KUKA KRL program: EPS_2_25856_SANMH_A_20250918023512.src

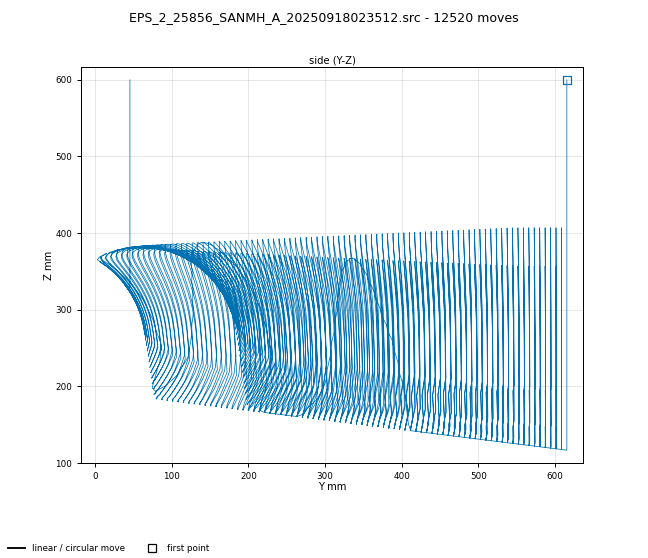
[picture p0: tool path of EPS_2_25856_SANMH_A_20250918023512.src, 12520 of 12522 moves have a stored position in this frame; points joined in program order, loops and branches not executed]
&ACCESS RVP
&REL 4
&COMMENT QRS 19112012
&PARAM EDITMASK = *
DEF PART()
EXT BAS (BAS_COMMAND :IN,REAL :IN )
INT I
BAS (#INITMOV,0 )

;KUKA QRS Post kuka4.cps  Date:22-06-2017 !

File_ID=2850

QRS_PRE_INIT()

;Init var - Until changes are made in qrs_pre_init
Outlet_Square_prg=0
Inlet_1_Square_prg=0
Inlet_2_Square_prg=0
Inlet_3_Square_prg=0
Inlet_4_Square_prg=0
Inlet_5_Square_prg=0

Outlet_1={X 0.000, Y 546.330, Z 306.500, B 0.000, E1 0.000 }
Inlet_1={X 0.000, Y 549.890, Z 256.500, B 0.000, E1 218.000 }
Outlet_1_type=201
Inlet_1_type=201
;QRS#1=Sidecore dimensions
;QRS#2=200-8" PVC SDR 35
;QRS#3=200-8" PVC SDR 35
;QRS#4=
;QRS#5=
;QRS#6=
;QRS#7=
;QRS#8=
;QRS#9=12-08 PSX
;QRS#10=12-08 PSX
;QRS#11=
;QRS#12=
;QRS#13=
;QRS#14=
;QRS#15=
;QRS#16=1220x127x686 2,25'
;QRS#17=EPS Height
;QRS#18=407
;QRS#19=*
;QRS#20= UPDATED VERSION 22-06-2017
;QRS#21=*
Outlet_Square=0100
Inlet_1_Square=0100
Inlet_2_Square=0
Inlet_3_Square=0
Inlet_4_Square=0
Inlet_5_Square=0
Mill_Square=1
Outlet_Square_Prg=204
Inlet_1_Square_prg=204

QRS_INIT()

$ADVANCE=5

; T1
PTP {E1 173.606,E2 173.606}
PTP {X 0,Y 615.506,A -85,B 0,C 180,E1 173.606,E2 173.606,E3 0,E4 0,E5 0,E6 0}
QRS_SPEED_INIT()
LIN {X 0,Y 615.506,Z 600,A -85,B 0,C 180,E1 173.606,E2 173.606,E3 0,E4 0,E5 0,E6 0} C_VEL
LIN {X 0,Y 615.506,Z 126.869,A -85,B 0,C 180,E1 173.606,E2 173.606} C_VEL
LIN {X 0,Y 615.506,Z 118.698,A -85,B 0,C 180,E1 173.606,E2 173.606} C_VEL
LIN {X 0,Y 615.487,Z 116.698,A -85,B 0,C 180,E1 173.42,E2 173.42} C_VEL
LIN {X 0,Y 615.471,Z 116.691,A -85,B 0,C 180,E1 170.801,E2 170.801} C_VEL
LIN {X 0,Y 615.488,Z 116.684,A -85,B 0,C 180,E1 168.14,E2 168.14} C_VEL
LIN {X 0,Y 615.489,Z 116.702,A -85,B 0,C 180,E1 165.451,E2 165.451} C_VEL
LIN {X 0,Y 615.476,Z 116.686,A -85,B 0,C 180,E1 162.73,E2 162.73} C_VEL
LIN {X 0,Y 615.48,Z 116.692,A -85,B 0,C 180,E1 159.967,E2 159.967} C_VEL
LIN {X 0,Y 615.492,Z 116.701,A -85,B 0,C 180,E1 157.652,E2 157.652} C_VEL
LIN {X 0,Y 615.473,Z 116.688,A -85,B 0,C 180,E1 155.008,E2 155.008} C_VEL
LIN {X 0,Y 615.481,Z 116.684,A -85,B 0,C 180,E1 152.823,E2 152.823} C_VEL
LIN {X 0,Y 615.482,Z 116.69,A -85,B 0,C 180,E1 150.206,E2 150.206} C_VEL
LIN {X 0,Y 615.48,Z 116.695,A -85,B 0,C 180,E1 147.543,E2 147.543} C_VEL
LIN {X 0,Y 615.475,Z 116.687,A -85,B 0,C 180,E1 145.185,E2 145.185} C_VEL
LIN {X 0,Y 615.493,Z 116.682,A -85,B 0,C 180,E1 142.759,E2 142.759} C_VEL
LIN {X 0,Y 615.494,Z 116.699,A -85,B 0,C 180,E1 139.91,E2 139.91} C_VEL
LIN {X 0,Y 615.488,Z 116.683,A -85,B 0,C 180,E1 136.952,E2 136.952} C_VEL
LIN {X 0,Y 615.49,Z 116.699,A -85,B 0,C 180,E1 133.998,E2 133.998} C_VEL
LIN {X 0,Y 615.487,Z 116.683,A -85,B 0,C 180,E1 131.095,E2 131.095} C_VEL
LIN {X 0,Y 615.487,Z 116.697,A -85,B 0,C 180,E1 128.068,E2 128.068} C_VEL
LIN {X 0,Y 615.473,Z 116.688,A -85,B 0,C 180,E1 125.616,E2 125.616} C_VEL
LIN {X 0,Y 615.487,Z 116.683,A -85,B 0,C 180,E1 123.236,E2 123.236} C_VEL
LIN {X 0,Y 615.481,Z 116.688,A -85,B 0,C 180,E1 120.92,E2 120.92} C_VEL
LIN {X 0,Y 615.497,Z 116.699,A -85,B 0,C 180,E1 118.453,E2 118.453} C_VEL
LIN {X 0,Y 615.485,Z 116.683,A -85,B 0,C 180,E1 115.569,E2 115.569} C_VEL
LIN {X 0,Y 615.482,Z 116.694,A -85,B 0,C 180,E1 112.844,E2 112.844} C_VEL
LIN {X 0,Y 615.488,Z 116.702,A -85,B 0,C 180,E1 110.558,E2 110.558} C_VEL
LIN {X 0,Y 615.478,Z 116.687,A -85,B 0,C 180,E1 107.957,E2 107.957} C_VEL
LIN {X 0,Y 615.479,Z 116.689,A -85,B 0,C 180,E1 105.226,E2 105.226} C_VEL
LIN {X 0,Y 615.485,Z 116.696,A -85,B 0,C 180,E1 102.53,E2 102.53} C_VEL
LIN {X 0,Y 615.493,Z 116.681,A -85,B 0,C 180,E1 99.862,E2 99.862} C_VEL
LIN {X 0,Y 615.48,Z 116.693,A -85,B 0,C 180,E1 97.215,E2 97.215} C_VEL
LIN {X 0,Y 615.48,Z 116.694,A -85,B 0,C 180,E1 94.584,E2 94.584} C_VEL
LIN {X 0,Y 615.5,Z 116.68,A -85,B 0,C 180,E1 91.963,E2 91.963} C_VEL
LIN {X 0,Y 615.48,Z 116.693,A -85,B 0,C 180,E1 89.345,E2 89.345} C_VEL
LIN {X 0,Y 615.48,Z 116.693,A -85,B 0,C 180,E1 86.727,E2 86.727} C_VEL
LIN {X 0,Y 615.498,Z 116.68,A -85,B 0,C 180,E1 84.101,E2 84.101} C_VEL
LIN {X 0,Y 615.481,Z 116.694,A -85,B 0,C 180,E1 81.463,E2 81.463} C_VEL
LIN {X 0,Y 615.477,Z 116.692,A -85,B 0,C 180,E1 78.806,E2 78.806} C_VEL
LIN {X 0,Y 615.483,Z 116.685,A -85,B 0,C 180,E1 76.067,E2 76.067} C_VEL
LIN {X 0,Y 615.494,Z 116.699,A -85,B 0,C 180,E1 73.413,E2 73.413} C_VEL
LIN {X 0,Y 615.485,Z 116.685,A -85,B 0,C 180,E1 70.662,E2 70.662} C_VEL
LIN {X 0,Y 615.476,Z 116.819,A -85,B 0,C 180,E1 69.966,E2 69.966} C_VEL
LIN {X 0,Y 615.473,Z 131.445,A -85,B 0,C 180,E1 67.404,E2 67.404} C_VEL
LIN {X 0,Y 615.472,Z 146.428,A -85,B 0,C 180,E1 64.808,E2 64.808} C_VEL
LIN {X 0,Y 615.434,Z 253.444,A -85,B 0,C 180,E1 63.534,E2 63.534} C_VEL
LIN {X 0,Y 615.441,Z 266.025,A -85,B 0,C 180,E1 63.256,E2 63.256} C_VEL
LIN {X 0,Y 615.475,Z 279.168,A -85,B 0,C 180,E1 62.822,E2 62.822} C_VEL
LIN {X 0,Y 615.472,Z 291.37,A -85,B 0,C 180,E1 62.269,E2 62.269} C_VEL
LIN {X 0,Y 615.477,Z 302.53,A -85,B 0,C 180,E1 61.617,E2 61.617} C_VEL
LIN {X 0,Y 615.5,Z 312.724,A -85,B 0,C 180,E1 60.875,E2 60.875} C_VEL
LIN {X 0,Y 615.498,Z 322.222,A -85,B 0,C 180,E1 60.021,E2 60.021} C_VEL
LIN {X 0,Y 615.497,Z 330.704,A -85,B 0,C 180,E1 59.08,E2 59.08} C_VEL
LIN {X 0,Y 615.498,Z 337.512,A -85,B 0,C 180,E1 58.153,E2 58.153} C_VEL
LIN {X 0,Y 615.495,Z 343.437,A -85,B 0,C 180,E1 57.154,E2 57.154} C_VEL
LIN {X 0,Y 615.495,Z 348.788,A -85,B 0,C 180,E1 55.978,E2 55.978} C_VEL
LIN {X 0,Y 615.497,Z 352.664,A -85,B 0,C 180,E1 54.786,E2 54.786} C_VEL
LIN {X 0,Y 615.494,Z 355.18,A -85,B 0,C 180,E1 53.575,E2 53.575} C_VEL
LIN {X 0,Y 615.496,Z 356.068,A -85,B 0,C 180,E1 52.758,E2 52.758} C_VEL
LIN {X 0,Y 615.494,Z 356.387,A -85,B 0,C 180,E1 51.931,E2 51.931} C_VEL
LIN {X 0,Y 615.495,Z 355.914,A -85,B 0,C 180,E1 50.936,E2 50.936} C_VEL
LIN {X 0,Y 615.496,Z 354.47,A -85,B 0,C 180,E1 49.909,E2 49.909} C_VEL
LIN {X 0,Y 615.494,Z 352.075,A -85,B 0,C 180,E1 48.904,E2 48.904} C_VEL
LIN {X 0,Y 615.497,Z 348.737,A -85,B 0,C 180,E1 47.918,E2 47.918} C_VEL
LIN {X 0,Y 615.498,Z 343.434,A -85,B 0,C 180,E1 46.756,E2 46.756} C_VEL
LIN {X 0,Y 615.494,Z 336.828,A -85,B 0,C 180,E1 45.655,E2 45.655} C_VEL
LIN {X 0,Y 615.495,Z 329.928,A -85,B 0,C 180,E1 44.735,E2 44.735} C_VEL
LIN {X 0,Y 615.498,Z 321.427,A -85,B 0,C 180,E1 43.808,E2 43.808} C_VEL
LIN {X 0,Y 615.499,Z 311.77,A -85,B 0,C 180,E1 42.96,E2 42.96} C_VEL
LIN {X 0,Y 615.47,Z 301.331,A -85,B 0,C 180,E1 42.215,E2 42.215} C_VEL
LIN {X 0,Y 615.466,Z 291.064,A -85,B 0,C 180,E1 41.625,E2 41.625} C_VEL
LIN {X 0,Y 615.486,Z 279.307,A -85,B 0,C 180,E1 41.094,E2 41.094} C_VEL
LIN {X 0,Y 615.456,Z 266.543,A -85,B 0,C 180,E1 40.669,E2 40.669} C_VEL
LIN {X 0,Y 615.445,Z 253.621,A -85,B 0,C 180,E1 40.379,E2 40.379} C_VEL
LIN {X 0,Y 615.497,Z 146.435,A -85,B 0,C 180,E1 39.104,E2 39.104} C_VEL
LIN {X 0,Y 615.48,Z 130.975,A -85,B 0,C 180,E1 36.425,E2 36.425} C_VEL
LIN {X 0,Y 615.465,Z 116.691,A -85,B 0,C 180,E1 33.9,E2 33.9} C_VEL
LIN {X 0,Y 615.491,Z 116.688,A -85,B 0,C 180,E1 31.086,E2 31.086} C_VEL
LIN {X 0,Y 615.475,Z 116.697,A -85,B 0,C 180,E1 28.447,E2 28.447} C_VEL
LIN {X 0,Y 615.472,Z 116.687,A -85,B 0,C 180,E1 25.716,E2 25.716} C_VEL
LIN {X 0,Y 615.483,Z 116.701,A -85,B 0,C 180,E1 22.844,E2 22.844} C_VEL
LIN {X 0,Y 615.46,Z 116.695,A -85,B 0,C 180,E1 20.549,E2 20.549} C_VEL
LIN {X 0,Y 615.464,Z 116.689,A -85,B 0,C 180,E1 17.957,E2 17.957} C_VEL
LIN {X 0,Y 615.492,Z 116.701,A -85,B 0,C 180,E1 15.225,E2 15.225} C_VEL
LIN {X 0,Y 615.446,Z 116.694,A -85,B 0,C 180,E1 12.531,E2 12.531} C_VEL
LIN {X 0,Y 615.49,Z 116.688,A -85,B 0,C 180,E1 9.862,E2 9.862} C_VEL
LIN {X 0,Y 615.467,Z 116.698,A -85,B 0,C 180,E1 7.216,E2 7.216} C_VEL
LIN {X 0,Y 615.462,Z 116.698,A -85,B 0,C 180,E1 5.241,E2 5.241} C_VEL
LIN {X 0,Y 615.438,Z 116.694,A -85,B 0,C 180,E1 2.618,E2 2.618} C_VEL
LIN {X 0,Y 615.487,Z 116.695,A -85,B 0,C 180,E1 0,E2 0} C_VEL
LIN {X 0,Y 615.446,Z 116.698,A -85,B 0,C 180,E1 -2.618,E2 -2.618} C_VEL
LIN {X 0,Y 615.442,Z 116.699,A -85,B 0,C 180,E1 -4.585,E2 -4.585} C_VEL
LIN {X 0,Y 615.438,Z 116.699,A -85,B 0,C 180,E1 -6.558,E2 -6.558} C_VEL
LIN {X 0,Y 615.433,Z 116.699,A -85,B 0,C 180,E1 -8.538,E2 -8.538} C_VEL
LIN {X 0,Y 615.42,Z 116.698,A -85,B 0,C 180,E1 -10.853,E2 -10.853} C_VEL
LIN {X 0,Y 615.437,Z 116.699,A -85,B 0,C 180,E1 -13.203,E2 -13.203} C_VEL
LIN {X 0,Y 615.464,Z 116.7,A -85,B 0,C 180,E1 -15.906,E2 -15.906} C_VEL
LIN {X 0,Y 615.414,Z 116.7,A -85,B 0,C 180,E1 -18.649,E2 -18.649} C_VEL
LIN {X 0,Y 615.495,Z 116.7,A -85,B 0,C 180,E1 -21.432,E2 -21.432} C_VEL
LIN {X 0,Y 615.422,Z 116.698,A -85,B 0,C 180,E1 -24.275,E2 -24.275} C_VEL
LIN {X 0,Y 615.424,Z 116.698,A -85,B 0,C 180,E1 -26.447,E2 -26.447} C_VEL
LIN {X 0,Y 615.483,Z 116.696,A -85,B 0,C 180,E1 -29.407,E2 -29.407} C_VEL
LIN {X 0,Y 615.452,Z 116.694,A -85,B 0,C 180,E1 -31.688,E2 -31.688} C_VEL
LIN {X 0,Y 615.433,Z 116.696,A -85,B 0,C 180,E1 -34.026,E2 -34.026} C_VEL
LIN {X 0,Y 615.488,Z 116.701,A -85,B 0,C 180,E1 -36.936,E2 -36.936} C_VEL
LIN {X 0,Y 615.44,Z 116.694,A -85,B 0,C 180,E1 -39.754,E2 -39.754} C_VEL
LIN {X 0,Y 615.461,Z 116.698,A -85,B 0,C 180,E1 -42.356,E2 -42.356} C_VEL
LIN {X 0,Y 615.491,Z 116.688,A -85,B 0,C 180,E1 -45.069,E2 -45.069} C_VEL
LIN {X 0,Y 615.447,Z 116.693,A -85,B 0,C 180,E1 -47.643,E2 -47.643} C_VEL
LIN {X 0,Y 615.479,Z 116.699,A -85,B 0,C 180,E1 -50.249,E2 -50.249} C_VEL
LIN {X 0,Y 615.474,Z 116.688,A -85,B 0,C 180,E1 -53.066,E2 -53.066} C_VEL
LIN {X 0,Y 615.457,Z 116.69,A -85,B 0,C 180,E1 -55.304,E2 -55.304} C_VEL
LIN {X 0,Y 615.461,Z 116.695,A -85,B 0,C 180,E1 -57.674,E2 -57.674} C_VEL
LIN {X 0,Y 615.489,Z 116.687,A -85,B 0,C 180,E1 -60.593,E2 -60.593} C_VEL
LIN {X 0,Y 615.468,Z 116.688,A -85,B 0,C 180,E1 -62.959,E2 -62.959} C_VEL
LIN {X 0,Y 615.482,Z 116.7,A -85,B 0,C 180,E1 -65.727,E2 -65.727} C_VEL
LIN {X 0,Y 615.464,Z 116.819,A -85,B 0,C 180,E1 -67.065,E2 -67.065} C_VEL
LIN {X 0,Y 615.465,Z 136.769,A -85,B 0,C 180,E1 -69.706,E2 -69.706} C_VEL
LIN {X 0,Y 615.485,Z 158.666,A -85,B 0,C 180,E1 -72.558,E2 -72.558} C_VEL
LIN {X 0,Y 615.469,Z 179.888,A -85,B 0,C 180,E1 -75.281,E2 -75.281} C_VEL
LIN {X 0,Y 615.452,Z 194.297,A -85,B 0,C 180,E1 -77.112,E2 -77.112} C_VEL
LIN {X 0,Y 615.488,Z 302.807,A -85,B 0,C 180,E1 -78.41,E2 -78.41} C_VEL
LIN {X 0,Y 615.477,Z 315.331,A -85,B 0,C 180,E1 -78.681,E2 -78.681} C_VEL
LIN {X 0,Y 615.488,Z 328.619,A -85,B 0,C 180,E1 -79.113,E2 -79.113} C_VEL
LIN {X 0,Y 615.477,Z 340.471,A -85,B 0,C 180,E1 -79.639,E2 -79.639} C_VEL
LIN {X 0,Y 615.494,Z 351.988,A -85,B 0,C 180,E1 -80.303,E2 -80.303} C_VEL
LIN {X 0,Y 615.499,Z 362.336,A -85,B 0,C 180,E1 -81.049,E2 -81.049} C_VEL
LIN {X 0,Y 615.497,Z 370.807,A -85,B 0,C 180,E1 -81.794,E2 -81.794} C_VEL
LIN {X 0,Y 615.498,Z 378.603,A -85,B 0,C 180,E1 -82.619,E2 -82.619} C_VEL
LIN {X 0,Y 615.496,Z 386.2,A -85,B 0,C 180,E1 -83.608,E2 -83.608} C_VEL
LIN {X 0,Y 615.498,Z 393.202,A -85,B 0,C 180,E1 -84.759,E2 -84.759} C_VEL
LIN {X 0,Y 615.494,Z 397.85,A -85,B 0,C 180,E1 -85.743,E2 -85.743} C_VEL
LIN {X 0,Y 615.494,Z 401.397,A -85,B 0,C 180,E1 -86.727,E2 -86.727} C_VEL
LIN {X 0,Y 615.497,Z 403.232,A -85,B 0,C 180,E1 -87.382,E2 -87.382} C_VEL
LIN {X 0,Y 615.5,Z 404.607,A -85,B 0,C 180,E1 -88.037,E2 -88.037} C_VEL
LIN {X 0,Y 615.496,Z 406.173,A -85,B 0,C 180,E1 -89.345,E2 -89.345} C_VEL
LIN {X 0,Y 615.494,Z 406.389,A -85,B 0,C 180,E1 -90,E2 -90} C_VEL
LIN {X 0,Y 615.495,Z 405.58,A -85,B 0,C 180,E1 -91.308,E2 -91.308} C_VEL
LIN {X 0,Y 615.5,Z 404.608,A -85,B 0,C 180,E1 -91.963,E2 -91.963} C_VEL
LIN {X 0,Y 615.497,Z 403.234,A -85,B 0,C 180,E1 -92.617,E2 -92.617} C_VEL
LIN {X 0,Y 615.496,Z 400.351,A -85,B 0,C 180,E1 -93.6,E2 -93.6} C_VEL
LIN {X 0,Y 615.498,Z 396.443,A -85,B 0,C 180,E1 -94.584,E2 -94.584} C_VEL
LIN {X 0,Y 615.499,Z 391.407,A -85,B 0,C 180,E1 -95.569,E2 -95.569} C_VEL
LIN {X 0,Y 615.497,Z 384.87,A -85,B 0,C 180,E1 -96.583,E2 -96.583} C_VEL
LIN {X 0,Y 615.497,Z 377.136,A -85,B 0,C 180,E1 -97.545,E2 -97.545} C_VEL
LIN {X 0,Y 615.498,Z 369.049,A -85,B 0,C 180,E1 -98.371,E2 -98.371} C_VEL
LIN {X 0,Y 615.499,Z 359.172,A -85,B 0,C 180,E1 -99.198,E2 -99.198} C_VEL
LIN {X 0,Y 615.488,Z 347.988,A -85,B 0,C 180,E1 -99.945,E2 -99.945} C_VEL
LIN {X 0,Y 615.482,Z 337.031,A -85,B 0,C 180,E1 -100.527,E2 -100.527} C_VEL
LIN {X 0,Y 615.48,Z 324.496,A -85,B 0,C 180,E1 -101.04,E2 -101.04} C_VEL
LIN {X 0,Y 615.479,Z 312.083,A -85,B 0,C 180,E1 -101.401,E2 -101.401} C_VEL
LIN {X 0,Y 615.493,Z 298.491,A -85,B 0,C 180,E1 -101.651,E2 -101.651} C_VEL
LIN {X 0,Y 615.452,Z 194.304,A -85,B 0,C 180,E1 -102.887,E2 -102.887} C_VEL
LIN {X 0,Y 615.494,Z 171.936,A -85,B 0,C 180,E1 -105.735,E2 -105.735} C_VEL
LIN {X 0,Y 615.456,Z 151.013,A -85,B 0,C 180,E1 -108.435,E2 -108.435} C_VEL
LIN {X 0,Y 615.488,Z 130.785,A -85,B 0,C 180,E1 -111.08,E2 -111.08} C_VEL
LIN {X 0,Y 615.465,Z 116.689,A -85,B 0,C 180,E1 -112.978,E2 -112.978} C_VEL
LIN {X 0,Y 615.489,Z 116.689,A -85,B 0,C 180,E1 -115.715,E2 -115.715} C_VEL
LIN {X 0,Y 615.469,Z 116.696,A -85,B 0,C 180,E1 -118.447,E2 -118.447} C_VEL
LIN {X 0,Y 615.479,Z 116.684,A -85,B 0,C 180,E1 -121.084,E2 -121.084} C_VEL
LIN {X 0,Y 615.492,Z 116.701,A -85,B 0,C 180,E1 -124.021,E2 -124.021} C_VEL
LIN {X 0,Y 615.478,Z 116.685,A -85,B 0,C 180,E1 -126.935,E2 -126.935} C_VEL
LIN {X 0,Y 615.491,Z 116.698,A -85,B 0,C 180,E1 -129.749,E2 -129.749} C_VEL
LIN {X 0,Y 615.466,Z 116.692,A -85,B 0,C 180,E1 -132.354,E2 -132.354} C_VEL
LIN {X 0,Y 615.496,Z 116.683,A -85,B 0,C 180,E1 -135.067,E2 -135.067} C_VEL
LIN {X 0,Y 615.481,Z 116.697,A -85,B 0,C 180,E1 -137.92,E2 -137.92} C_VEL
LIN {X 0,Y 615.465,Z 116.691,A -85,B 0,C 180,E1 -140.248,E2 -140.248} C_VEL
LIN {X 0,Y 615.488,Z 116.687,A -85,B 0,C 180,E1 -143.063,E2 -143.063} C_VEL
LIN {X 0,Y 615.47,Z 116.693,A -85,B 0,C 180,E1 -145.977,E2 -145.977} C_VEL
LIN {X 0,Y 615.469,Z 116.688,A -85,B 0,C 180,E1 -148.313,E2 -148.313} C_VEL
LIN {X 0,Y 615.486,Z 116.683,A -85,B 0,C 180,E1 -150.593,E2 -150.593} C_VEL
LIN {X 0,Y 615.481,Z 116.698,A -85,B 0,C 180,E1 -153.555,E2 -153.555} C_VEL
LIN {X 0,Y 615.485,Z 116.684,A -85,B 0,C 180,E1 -156.443,E2 -156.443} C_VEL
LIN {X 0,Y 615.481,Z 116.698,A -85,B 0,C 180,E1 -159.444,E2 -159.444} C_VEL
LIN {X 0,Y 615.473,Z 116.686,A -85,B 0,C 180,E1 -162.042,E2 -162.042} C_VEL
LIN {X 0,Y 615.485,Z 116.691,A -85,B 0,C 180,E1 -164.774,E2 -164.774} C_VEL
LIN {X 0,Y 615.471,Z 116.695,A -85,B 0,C 180,E1 -167.469,E2 -167.469} C_VEL
LIN {X 0,Y 615.492,Z 116.682,A -85,B 0,C 180,E1 -170.138,E2 -170.138} C_VEL
LIN {X 0,Y 615.489,Z 116.695,A -85,B 0,C 180,E1 -172.784,E2 -172.784} C_VEL
LIN {X 0,Y 615.471,Z 116.692,A -85,B 0,C 180,E1 -175.415,E2 -175.415} C_VEL
LIN {X 0,Y 615.5,Z 116.68,A -85,B 0,C 180,E1 -178.037,E2 -178.037} C_VEL
LIN {X 0,Y 615.49,Z 116.696,A -85,B 0,C 180,E1 -180.654,E2 -180.654} C_VEL
LIN {X 0,Y 615.471,Z 116.692,A -85,B 0,C 180,E1 -183.273,E2 -183.273} C_VEL
LIN {X 0,Y 615.498,Z 116.681,A -85,B 0,C 180,E1 -185.898,E2 -185.898} C_VEL
LIN {X 0,Y 615.487,Z 116.698,A -85,B 0,C 180,E1 -186.58,E2 -186.58} C_VEL
LIN {X 0,Y 614.8,Z 116.838,A -85,B 0,C 180,E1 -187.126,E2 -187.126} C_VEL
LIN {X 0,Y 611.955,Z 117.252,A -85,B 0,C 180,E1 -188.012,E2 -188.012} C_VEL
LIN {X 0,Y 609.565,Z 117.562,A -85,B 0,C 180,E1 -188.725,E2 -188.725} C_VEL
LIN {X 0,Y 608.538,Z 117.679,A -85,B 0,C 180,E1 -189.274,E2 -189.274} C_VEL
LIN {X 0,Y 608.453,Z 117.688,A -85,B 0,C 180,E1 -189.461,E2 -189.461} C_VEL
LIN {X 0,Y 608.464,Z 117.688,A -85,B 0,C 180,E1 -191.999,E2 -191.999} C_VEL
LIN {X 0,Y 608.474,Z 117.692,A -85,B 0,C 180,E1 -194.72,E2 -194.72} C_VEL
LIN {X 0,Y 608.445,Z 117.688,A -85,B 0,C 180,E1 -197.476,E2 -197.476} C_VEL
LIN {X 0,Y 608.461,Z 117.694,A -85,B 0,C 180,E1 -200.274,E2 -200.274} C_VEL
LIN {X 0,Y 608.455,Z 117.696,A -85,B 0,C 180,E1 -202.476,E2 -202.476} C_VEL
LIN {X 0,Y 608.449,Z 117.694,A -85,B 0,C 180,E1 -204.571,E2 -204.571} C_VEL
LIN {X 0,Y 608.473,Z 117.685,A -85,B 0,C 180,E1 -207.207,E2 -207.207} C_VEL
LIN {X 0,Y 608.467,Z 117.692,A -85,B 0,C 180,E1 -209.972,E2 -209.972} C_VEL
LIN {X 0,Y 608.455,Z 117.692,A -85,B 0,C 180,E1 -212.522,E2 -212.522} C_VEL
LIN {X 0,Y 608.436,Z 117.69,A -85,B 0,C 180,E1 -215.278,E2 -215.278} C_VEL
LIN {X 0,Y 608.471,Z 117.69,A -85,B 0,C 180,E1 -217.746,E2 -217.746} C_VEL
LIN {X 0,Y 608.45,Z 117.693,A -85,B 0,C 180,E1 -220.329,E2 -220.329} C_VEL
LIN {X 0,Y 608.453,Z 117.687,A -85,B 0,C 180,E1 -222.959,E2 -222.959} C_VEL
LIN {X 0,Y 608.464,Z 117.694,A -85,B 0,C 180,E1 -225.735,E2 -225.735} C_VEL
LIN {X 0,Y 608.457,Z 117.687,A -85,B 0,C 180,E1 -228.658,E2 -228.658} C_VEL
LIN {X 0,Y 608.468,Z 117.69,A -85,B 0,C 180,E1 -231.412,E2 -231.412} C_VEL
LIN {X 0,Y 608.471,Z 117.692,A -85,B 0,C 180,E1 -233.951,E2 -233.951} C_VEL
LIN {X 0,Y 608.458,Z 117.688,A -85,B 0,C 180,E1 -236.329,E2 -236.329} C_VEL
LIN {X 0,Y 608.473,Z 117.685,A -85,B 0,C 180,E1 -238.727,E2 -238.727} C_VEL
LIN {X 0,Y 608.476,Z 117.691,A -85,B 0,C 180,E1 -241.379,E2 -241.379} C_VEL
LIN {X 0,Y 608.467,Z 117.686,A -85,B 0,C 180,E1 -244.279,E2 -244.279} C_VEL
LIN {X 0,Y 608.448,Z 117.69,A -85,B 0,C 180,E1 -246.876,E2 -246.876} C_VEL
LIN {X 0,Y 608.467,Z 117.695,A -85,B 0,C 180,E1 -249.32,E2 -249.32} C_VEL
LIN {X 0,Y 608.446,Z 117.692,A -85,B 0,C 180,E1 -251.828,E2 -251.828} C_VEL
LIN {X 0,Y 608.465,Z 117.687,A -85,B 0,C 180,E1 -254.594,E2 -254.594} C_VEL
LIN {X 0,Y 608.473,Z 117.695,A -85,B 0,C 180,E1 -257.323,E2 -257.323} C_VEL
LIN {X 0,Y 608.461,Z 117.687,A -85,B 0,C 180,E1 -260.023,E2 -260.023} C_VEL
LIN {X 0,Y 608.459,Z 117.69,A -85,B 0,C 180,E1 -262.701,E2 -262.701} C_VEL
LIN {X 0,Y 608.46,Z 117.69,A -85,B 0,C 180,E1 -264.698,E2 -264.698} C_VEL
LIN {X 0,Y 608.472,Z 117.69,A -85,B 0,C 180,E1 -267.352,E2 -267.352} C_VEL
LIN {X 0,Y 608.477,Z 117.684,A -85,B 0,C 180,E1 -270,E2 -270} C_VEL
LIN {X 0,Y 608.472,Z 117.69,A -85,B 0,C 180,E1 -272.648,E2 -272.648} C_VEL
LIN {X 0,Y 608.461,Z 117.69,A -85,B 0,C 180,E1 -275.302,E2 -275.302} C_VEL
LIN {X 0,Y 608.477,Z 117.685,A -85,B 0,C 180,E1 -277.967,E2 -277.967} C_VEL
LIN {X 0,Y 608.469,Z 117.693,A -85,B 0,C 180,E1 -280.958,E2 -280.958} C_VEL
LIN {X 0,Y 608.458,Z 117.688,A -85,B 0,C 180,E1 -283.357,E2 -283.357} C_VEL
LIN {X 0,Y 608.458,Z 117.689,A -85,B 0,C 180,E1 -286.094,E2 -286.094} C_VEL
LIN {X 0,Y 608.456,Z 117.694,A -85,B 0,C 180,E1 -288.87,E2 -288.87} C_VEL
LIN {X 0,Y 608.457,Z 117.733,A -85,B 0,C 180,E1 -289.966,E2 -289.966} C_VEL
LIN {X 0,Y 608.457,Z 131.94,A -85,B 0,C 180,E1 -292.477,E2 -292.477} C_VEL
LIN {X 0,Y 608.428,Z 146.561,A -85,B 0,C 180,E1 -295.028,E2 -295.028} C_VEL
LIN {X 0,Y 608.57,Z 154.029,A -85,B 0,C 180,E1 -295.136,E2 -295.136} C_VEL
LIN {X 0,Y 608.493,Z 253.638,A -85,B 0,C 180,E1 -296.333,E2 -296.333} C_VEL
LIN {X 0,Y 608.49,Z 266.859,A -85,B 0,C 180,E1 -296.634,E2 -296.634} C_VEL
LIN {X 0,Y 608.515,Z 279.85,A -85,B 0,C 180,E1 -297.074,E2 -297.074} C_VEL
LIN {X 0,Y 608.476,Z 291.511,A -85,B 0,C 180,E1 -297.61,E2 -297.61} C_VEL
LIN {X 0,Y 608.462,Z 302.667,A -85,B 0,C 180,E1 -298.267,E2 -298.267} C_VEL
LIN {X 0,Y 608.485,Z 312.956,A -85,B 0,C 180,E1 -299.019,E2 -299.019} C_VEL
LIN {X 0,Y 608.483,Z 321.485,A -85,B 0,C 180,E1 -299.779,E2 -299.779} C_VEL
LIN {X 0,Y 608.459,Z 330.175,A -85,B 0,C 180,E1 -300.726,E2 -300.726} C_VEL
LIN {X 0,Y 608.463,Z 337.47,A -85,B 0,C 180,E1 -301.705,E2 -301.705} C_VEL
LIN {X 0,Y 608.432,Z 342.458,A -85,B 0,C 180,E1 -302.519,E2 -302.519} C_VEL
LIN {X 0,Y 608.425,Z 348.328,A -85,B 0,C 180,E1 -303.729,E2 -303.729} C_VEL
LIN {X 0,Y 608.427,Z 352.487,A -85,B 0,C 180,E1 -304.903,E2 -304.903} C_VEL
LIN {X 0,Y 608.421,Z 355.26,A -85,B 0,C 180,E1 -306.094,E2 -306.094} C_VEL
LIN {X 0,Y 608.435,Z 356.623,A -85,B 0,C 180,E1 -307.155,E2 -307.155} C_VEL
LIN {X 0,Y 608.42,Z 356.961,A -85,B 0,C 180,E1 -308.235,E2 -308.235} C_VEL
LIN {X 0,Y 608.418,Z 356.095,A -85,B 0,C 180,E1 -309.444,E2 -309.444} C_VEL
LIN {X 0,Y 608.433,Z 353.685,A -85,B 0,C 180,E1 -310.74,E2 -310.74} C_VEL
LIN {X 0,Y 608.45,Z 350.941,A -85,B 0,C 180,E1 -311.674,E2 -311.674} C_VEL
LIN {X 0,Y 608.442,Z 347.218,A -85,B 0,C 180,E1 -312.62,E2 -312.62} C_VEL
LIN {X 0,Y 608.453,Z 342.507,A -85,B 0,C 180,E1 -313.562,E2 -313.562} C_VEL
LIN {X 0,Y 608.459,Z 335.68,A -85,B 0,C 180,E1 -314.649,E2 -314.649} C_VEL
LIN {X 0,Y 608.469,Z 326.965,A -85,B 0,C 180,E1 -315.736,E2 -315.736} C_VEL
LIN {X 0,Y 608.476,Z 318.467,A -85,B 0,C 180,E1 -316.595,E2 -316.595} C_VEL
LIN {X 0,Y 608.478,Z 308.923,A -85,B 0,C 180,E1 -317.386,E2 -317.386} C_VEL
LIN {X 0,Y 608.475,Z 297.672,A -85,B 0,C 180,E1 -318.135,E2 -318.135} C_VEL
LIN {X 0,Y 608.513,Z 285.502,A -85,B 0,C 180,E1 -318.774,E2 -318.774} C_VEL
LIN {X 0,Y 608.513,Z 272.973,A -85,B 0,C 180,E1 -319.267,E2 -319.267} C_VEL
LIN {X 0,Y 608.5,Z 259.837,A -85,B 0,C 180,E1 -319.633,E2 -319.633} C_VEL
LIN {X 0,Y 608.505,Z 247.33,A -85,B 0,C 180,E1 -319.85,E2 -319.85} C_VEL
LIN {X 0,Y 608.462,Z 146.633,A -85,B 0,C 180,E1 -321.048,E2 -321.048} C_VEL
LIN {X 0,Y 608.473,Z 131.414,A -85,B 0,C 180,E1 -323.705,E2 -323.705} C_VEL
LIN {X 0,Y 608.448,Z 117.69,A -85,B 0,C 180,E1 -326.148,E2 -326.148} C_VEL
LIN {X 0,Y 608.449,Z 117.69,A -85,B 0,C 180,E1 -328.733,E2 -328.733} C_VEL
LIN {X 0,Y 608.469,Z 117.695,A -85,B 0,C 180,E1 -331.382,E2 -331.382} C_VEL
LIN {X 0,Y 608.431,Z 117.691,A -85,B 0,C 180,E1 -333.964,E2 -333.964} C_VEL
LIN {X 0,Y 608.449,Z 117.695,A -85,B 0,C 180,E1 -336.876,E2 -336.876} C_VEL
LIN {X 0,Y 608.45,Z 117.693,A -85,B 0,C 180,E1 -339.327,E2 -339.327} C_VEL
LIN {X 0,Y 608.425,Z 117.691,A -85,B 0,C 180,E1 -341.828,E2 -341.828} C_VEL
LIN {X 0,Y 608.472,Z 117.692,A -85,B 0,C 180,E1 -344.595,E2 -344.595} C_VEL
LIN {X 0,Y 608.423,Z 117.693,A -85,B 0,C 180,E1 -347.322,E2 -347.322} C_VEL
LIN {X 0,Y 608.452,Z 117.69,A -85,B 0,C 180,E1 -350.023,E2 -350.023} C_VEL
LIN {X 0,Y 608.438,Z 117.697,A -85,B 0,C 180,E1 -352.701,E2 -352.701} C_VEL
LIN {X 0,Y 608.446,Z 117.694,A -85,B 0,C 180,E1 -354.698,E2 -354.698} C_VEL
LIN {X 0,Y 608.435,Z 117.69,A -85,B 0,C 180,E1 -357.352,E2 -357.352} C_VEL
LIN {X 0,Y 608.478,Z 117.691,A -85,B 0,C 180,E1 -360,E2 -360} C_VEL
LIN {X 0,Y 608.44,Z 117.692,A -85,B 0,C 180,E1 -362.649,E2 -362.649} C_VEL
LIN {X 0,Y 608.42,Z 117.692,A -85,B 0,C 180,E1 -365.303,E2 -365.303} C_VEL
LIN {X 0,Y 608.471,Z 117.696,A -85,B 0,C 180,E1 -367.967,E2 -367.967} C_VEL
LIN {X 0,Y 608.407,Z 117.694,A -85,B 0,C 180,E1 -370.651,E2 -370.651} C_VEL
LIN {X 0,Y 608.427,Z 117.695,A -85,B 0,C 180,E1 -373.358,E2 -373.358} C_VEL
LIN {X 0,Y 608.423,Z 117.695,A -85,B 0,C 180,E1 -376.095,E2 -376.095} C_VEL
LIN {X 0,Y 608.401,Z 117.695,A -85,B 0,C 180,E1 -378.872,E2 -378.872} C_VEL
LIN {X 0,Y 608.453,Z 117.694,A -85,B 0,C 180,E1 -381.692,E2 -381.692} C_VEL
LIN {X 0,Y 608.411,Z 117.693,A -85,B 0,C 180,E1 -384.573,E2 -384.573} C_VEL
LIN {X 0,Y 608.473,Z 117.695,A -85,B 0,C 180,E1 -387.205,E2 -387.205} C_VEL
LIN {X 0,Y 608.41,Z 117.694,A -85,B 0,C 180,E1 -389.961,E2 -389.961} C_VEL
LIN {X 0,Y 608.423,Z 117.694,A -85,B 0,C 180,E1 -392.516,E2 -392.516} C_VEL
LIN {X 0,Y 608.423,Z 117.696,A -85,B 0,C 180,E1 -395.279,E2 -395.279} C_VEL
LIN {X 0,Y 608.439,Z 117.69,A -85,B 0,C 180,E1 -397.749,E2 -397.749} C_VEL
LIN {X 0,Y 608.438,Z 117.693,A -85,B 0,C 180,E1 -400.327,E2 -400.327} C_VEL
LIN {X 0,Y 608.463,Z 117.688,A -85,B 0,C 180,E1 -403.307,E2 -403.307} C_VEL
LIN {X 0,Y 608.444,Z 117.692,A -85,B 0,C 180,E1 -406.128,E2 -406.128} C_VEL
LIN {X 0,Y 608.459,Z 117.691,A -85,B 0,C 180,E1 -408.823,E2 -408.823} C_VEL
LIN {X 0,Y 608.447,Z 117.69,A -85,B 0,C 180,E1 -411.763,E2 -411.763} C_VEL
LIN {X 0,Y 608.446,Z 117.694,A -85,B 0,C 180,E1 -413.955,E2 -413.955} C_VEL
LIN {X 0,Y 608.455,Z 117.696,A -85,B 0,C 180,E1 -416.328,E2 -416.328} C_VEL
LIN {X 0,Y 608.449,Z 117.69,A -85,B 0,C 180,E1 -418.733,E2 -418.733} C_VEL
LIN {X 0,Y 608.453,Z 117.689,A -85,B 0,C 180,E1 -421.384,E2 -421.384} C_VEL
LIN {X 0,Y 608.44,Z 117.699,A -85,B 0,C 180,E1 -423.964,E2 -423.964} C_VEL
LIN {X 0,Y 608.472,Z 117.692,A -85,B 0,C 180,E1 -426.155,E2 -426.155} C_VEL
LIN {X 0,Y 608.468,Z 117.817,A -85,B 0,C 180,E1 -426.921,E2 -426.921} C_VEL
LIN {X 0,Y 608.585,Z 133.439,A -85,B 0,C 180,E1 -429.023,E2 -429.023} C_VEL
LIN {X 0,Y 608.522,Z 154.713,A -85,B 0,C 180,E1 -431.83,E2 -431.83} C_VEL
LIN {X 0,Y 608.49,Z 175.987,A -85,B 0,C 180,E1 -434.594,E2 -434.594} C_VEL
LIN {X 0,Y 608.45,Z 194.518,A -85,B 0,C 180,E1 -436.972,E2 -436.972} C_VEL
LIN {X 0,Y 608.547,Z 302.924,A -85,B 0,C 180,E1 -438.276,E2 -438.276} C_VEL
LIN {X 0,Y 608.512,Z 316.202,A -85,B 0,C 180,E1 -438.571,E2 -438.571} C_VEL
LIN {X 0,Y 608.514,Z 328.628,A -85,B 0,C 180,E1 -438.982,E2 -438.982} C_VEL
LIN {X 0,Y 608.499,Z 340.627,A -85,B 0,C 180,E1 -439.519,E2 -439.519} C_VEL
LIN {X 0,Y 608.484,Z 352.191,A -85,B 0,C 180,E1 -440.191,E2 -440.191} C_VEL
LIN {X 0,Y 608.485,Z 362.589,A -85,B 0,C 180,E1 -440.945,E2 -440.945} C_VEL
LIN {X 0,Y 608.475,Z 371.107,A -85,B 0,C 180,E1 -441.698,E2 -441.698} C_VEL
LIN {X 0,Y 608.471,Z 378.957,A -85,B 0,C 180,E1 -442.533,E2 -442.533} C_VEL
LIN {X 0,Y 608.461,Z 386.286,A -85,B 0,C 180,E1 -443.484,E2 -443.484} C_VEL
LIN {X 0,Y 608.451,Z 391.864,A -85,B 0,C 180,E1 -444.365,E2 -444.365} C_VEL
LIN {X 0,Y 608.432,Z 396.948,A -85,B 0,C 180,E1 -445.362,E2 -445.362} C_VEL
LIN {X 0,Y 608.449,Z 400.895,A -85,B 0,C 180,E1 -446.357,E2 -446.357} C_VEL
LIN {X 0,Y 608.425,Z 403.808,A -85,B 0,C 180,E1 -447.351,E2 -447.351} C_VEL
LIN {X 0,Y 608.445,Z 405.201,A -85,B 0,C 180,E1 -448.014,E2 -448.014} C_VEL
LIN {X 0,Y 608.438,Z 406.783,A -85,B 0,C 180,E1 -449.338,E2 -449.338} C_VEL
LIN {X 0,Y 608.434,Z 407,A -85,B 0,C 180,E1 -450,E2 -450} C_VEL
LIN {X 0,Y 608.448,Z 406.184,A -85,B 0,C 180,E1 -451.323,E2 -451.323} C_VEL
LIN {X 0,Y 608.445,Z 405.202,A -85,B 0,C 180,E1 -451.985,E2 -451.985} C_VEL
LIN {X 0,Y 608.425,Z 403.81,A -85,B 0,C 180,E1 -452.648,E2 -452.648} C_VEL
LIN {X 0,Y 608.449,Z 400.897,A -85,B 0,C 180,E1 -453.642,E2 -453.642} C_VEL
LIN {X 0,Y 608.432,Z 396.952,A -85,B 0,C 180,E1 -454.637,E2 -454.637} C_VEL
LIN {X 0,Y 608.438,Z 390.879,A -85,B 0,C 180,E1 -455.8,E2 -455.8} C_VEL
LIN {X 0,Y 608.462,Z 384.238,A -85,B 0,C 180,E1 -456.799,E2 -456.799} C_VEL
LIN {X 0,Y 608.456,Z 375.992,A -85,B 0,C 180,E1 -457.8,E2 -457.8} C_VEL
LIN {X 0,Y 608.472,Z 367.541,A -85,B 0,C 180,E1 -458.635,E2 -458.635} C_VEL
LIN {X 0,Y 608.479,Z 357.096,A -85,B 0,C 180,E1 -459.473,E2 -459.473} C_VEL
LIN {X 0,Y 608.489,Z 346.762,A -85,B 0,C 180,E1 -460.144,E2 -460.144} C_VEL
LIN {X 0,Y 608.519,Z 335.273,A -85,B 0,C 180,E1 -460.74,E2 -460.74} C_VEL
LIN {X 0,Y 608.528,Z 322.9,A -85,B 0,C 180,E1 -461.224,E2 -461.224} C_VEL
LIN {X 0,Y 608.544,Z 309.454,A -85,B 0,C 180,E1 -461.596,E2 -461.596} C_VEL
LIN {X 0,Y 608.553,Z 297.113,A -85,B 0,C 180,E1 -461.807,E2 -461.807} C_VEL
LIN {X 0,Y 608.438,Z 194.441,A -85,B 0,C 180,E1 -463.038,E2 -463.038} C_VEL
LIN {X 0,Y 608.51,Z 172.004,A -85,B 0,C 180,E1 -465.92,E2 -465.92} C_VEL
LIN {X 0,Y 608.5,Z 152.263,A -85,B 0,C 180,E1 -468.492,E2 -468.492} C_VEL
LIN {X 0,Y 608.566,Z 132.116,A -85,B 0,C 180,E1 -471.154,E2 -471.154} C_VEL
LIN {X 0,Y 608.465,Z 117.74,A -85,B 0,C 180,E1 -473.089,E2 -473.089} C_VEL
LIN {X 0,Y 608.475,Z 117.688,A -85,B 0,C 180,E1 -475.721,E2 -475.721} C_VEL
LIN {X 0,Y 608.442,Z 117.697,A -85,B 0,C 180,E1 -478.267,E2 -478.267} C_VEL
LIN {X 0,Y 608.465,Z 117.689,A -85,B 0,C 180,E1 -480.545,E2 -480.545} C_VEL
LIN {X 0,Y 608.451,Z 117.688,A -85,B 0,C 180,E1 -482.879,E2 -482.879} C_VEL
LIN {X 0,Y 608.436,Z 117.691,A -85,B 0,C 180,E1 -485.278,E2 -485.278} C_VEL
LIN {X 0,Y 608.469,Z 117.693,A -85,B 0,C 180,E1 -487.746,E2 -487.746} C_VEL
LIN {X 0,Y 608.439,Z 117.692,A -85,B 0,C 180,E1 -490.327,E2 -490.327} C_VEL
LIN {X 0,Y 608.477,Z 117.687,A -85,B 0,C 180,E1 -493.309,E2 -493.309} C_VEL
LIN {X 0,Y 608.464,Z 117.69,A -85,B 0,C 180,E1 -496.13,E2 -496.13} C_VEL
LIN {X 0,Y 608.453,Z 117.688,A -85,B 0,C 180,E1 -498.823,E2 -498.823} C_VEL
LIN {X 0,Y 608.46,Z 117.695,A -85,B 0,C 180,E1 -501.76,E2 -501.76} C_VEL
LIN {X 0,Y 608.441,Z 117.693,A -85,B 0,C 180,E1 -503.955,E2 -503.955} C_VEL
LIN {X 0,Y 608.442,Z 117.689,A -85,B 0,C 180,E1 -506.328,E2 -506.328} C_VEL
LIN {X 0,Y 608.447,Z 117.689,A -85,B 0,C 180,E1 -508.732,E2 -508.732} C_VEL
LIN {X 0,Y 608.472,Z 117.695,A -85,B 0,C 180,E1 -511.38,E2 -511.38} C_VEL
LIN {X 0,Y 608.438,Z 117.691,A -85,B 0,C 180,E1 -513.964,E2 -513.964} C_VEL
LIN {X 0,Y 608.453,Z 117.691,A -85,B 0,C 180,E1 -516.876,E2 -516.876} C_VEL
LIN {X 0,Y 608.465,Z 117.696,A -85,B 0,C 180,E1 -519.321,E2 -519.321} C_VEL
LIN {X 0,Y 608.439,Z 117.691,A -85,B 0,C 180,E1 -521.827,E2 -521.827} C_VEL
LIN {X 0,Y 608.468,Z 117.688,A -85,B 0,C 180,E1 -524.594,E2 -524.594} C_VEL
LIN {X 0,Y 608.464,Z 117.693,A -85,B 0,C 180,E1 -527.322,E2 -527.322} C_VEL
LIN {X 0,Y 608.458,Z 117.687,A -85,B 0,C 180,E1 -530.022,E2 -530.022} C_VEL
LIN {X 0,Y 608.466,Z 117.691,A -85,B 0,C 180,E1 -532.7,E2 -532.7} C_VEL
LIN {X 0,Y 608.467,Z 117.692,A -85,B 0,C 180,E1 -534.698,E2 -534.698} C_VEL
LIN {X 0,Y 608.464,Z 117.689,A -85,B 0,C 180,E1 -537.352,E2 -537.352} C_VEL
LIN {X 0,Y 608.477,Z 117.685,A -85,B 0,C 180,E1 -540,E2 -540} C_VEL
LIN {X 0,Y 608.477,Z 117.692,A -85,B 0,C 180,E1 -542.648,E2 -542.648} C_VEL
LIN {X 0,Y 608.453,Z 117.689,A -85,B 0,C 180,E1 -545.302,E2 -545.302} C_VEL
LIN {X 0,Y 608.479,Z 117.685,A -85,B 0,C 180,E1 -547.967,E2 -547.967} C_VEL
LIN {X 0,Y 608.453,Z 117.688,A -85,B 0,C 180,E1 -549.461,E2 -549.461} C_VEL
LIN {X 0,Y 607.784,Z 117.773,A -85,B 0,C 180,E1 -550.013,E2 -550.013} C_VEL
LIN {X 0,Y 604.934,Z 118.131,A -85,B 0,C 180,E1 -550.91,E2 -550.91} C_VEL
LIN {X 0,Y 602.528,Z 118.43,A -85,B 0,C 180,E1 -551.631,E2 -551.631} C_VEL
LIN {X 0,Y 601.494,Z 118.558,A -85,B 0,C 180,E1 -552.188,E2 -552.188} C_VEL
LIN {X 0,Y 601.41,Z 118.568,A -85,B 0,C 180,E1 -552.377,E2 -552.377} C_VEL
LIN {X 0,Y 601.427,Z 118.567,A -85,B 0,C 180,E1 -554.897,E2 -554.897} C_VEL
LIN {X 0,Y 601.428,Z 118.565,A -85,B 0,C 180,E1 -556.986,E2 -556.986} C_VEL
LIN {X 0,Y 601.403,Z 118.567,A -85,B 0,C 180,E1 -559.809,E2 -559.809} C_VEL
LIN {X 0,Y 601.408,Z 118.57,A -85,B 0,C 180,E1 -562.683,E2 -562.683} C_VEL
LIN {X 0,Y 601.399,Z 118.568,A -85,B 0,C 180,E1 -564.878,E2 -564.878} C_VEL
LIN {X 0,Y 601.418,Z 118.568,A -85,B 0,C 180,E1 -567.867,E2 -567.867} C_VEL
LIN {X 0,Y 601.425,Z 118.572,A -85,B 0,C 180,E1 -570.164,E2 -570.164} C_VEL
LIN {X 0,Y 601.418,Z 118.566,A -85,B 0,C 180,E1 -572.715,E2 -572.715} C_VEL
LIN {X 0,Y 601.39,Z 118.567,A -85,B 0,C 180,E1 -575.112,E2 -575.112} C_VEL
LIN {X 0,Y 601.433,Z 118.563,A -85,B 0,C 180,E1 -577.419,E2 -577.419} C_VEL
LIN {X 0,Y 601.409,Z 118.575,A -85,B 0,C 180,E1 -579.995,E2 -579.995} C_VEL
LIN {X 0,Y 601.408,Z 118.566,A -85,B 0,C 180,E1 -582.67,E2 -582.67} C_VEL
LIN {X 0,Y 601.421,Z 118.567,A -85,B 0,C 180,E1 -585.482,E2 -585.482} C_VEL
LIN {X 0,Y 601.423,Z 118.565,A -85,B 0,C 180,E1 -588.406,E2 -588.406} C_VEL
LIN {X 0,Y 601.435,Z 118.562,A -85,B 0,C 180,E1 -590.876,E2 -590.876} C_VEL
LIN {X 0,Y 601.439,Z 118.572,A -85,B 0,C 180,E1 -593.734,E2 -593.734} C_VEL
LIN {X 0,Y 601.424,Z 118.563,A -85,B 0,C 180,E1 -596.687,E2 -596.687} C_VEL
LIN {X 0,Y 601.426,Z 118.565,A -85,B 0,C 180,E1 -599.059,E2 -599.059} C_VEL
LIN {X 0,Y 601.435,Z 118.568,A -85,B 0,C 180,E1 -601.374,E2 -601.374} C_VEL
LIN {X 0,Y 601.401,Z 118.575,A -85,B 0,C 180,E1 -603.637,E2 -603.637} C_VEL
LIN {X 0,Y 601.416,Z 118.564,A -85,B 0,C 180,E1 -606.59,E2 -606.59} C_VEL
LIN {X 0,Y 601.429,Z 118.572,A -85,B 0,C 180,E1 -609.479,E2 -609.479} C_VEL
LIN {X 0,Y 601.392,Z 118.567,A -85,B 0,C 180,E1 -612.312,E2 -612.312} C_VEL
LIN {X 0,Y 601.41,Z 118.565,A -85,B 0,C 180,E1 -614.409,E2 -614.409} C_VEL
LIN {X 0,Y 601.417,Z 118.573,A -85,B 0,C 180,E1 -617.172,E2 -617.172} C_VEL
LIN {X 0,Y 601.437,Z 118.562,A -85,B 0,C 180,E1 -619.905,E2 -619.905} C_VEL
LIN {X 0,Y 601.437,Z 118.564,A -85,B 0,C 180,E1 -622.615,E2 -622.615} C_VEL
LIN {X 0,Y 601.418,Z 118.571,A -85,B 0,C 180,E1 -625.308,E2 -625.308} C_VEL
LIN {X 0,Y 601.438,Z 118.561,A -85,B 0,C 180,E1 -627.991,E2 -627.991} C_VEL
LIN {X 0,Y 601.446,Z 118.565,A -85,B 0,C 180,E1 -630.67,E2 -630.67} C_VEL
LIN {X 0,Y 601.426,Z 118.566,A -85,B 0,C 180,E1 -633.35,E2 -633.35} C_VEL
LIN {X 0,Y 601.441,Z 118.561,A -85,B 0,C 180,E1 -636.037,E2 -636.037} C_VEL
LIN {X 0,Y 601.432,Z 118.571,A -85,B 0,C 180,E1 -638.738,E2 -638.738} C_VEL
LIN {X 0,Y 601.431,Z 118.563,A -85,B 0,C 180,E1 -641.459,E2 -641.459} C_VEL
LIN {X 0,Y 601.417,Z 118.567,A -85,B 0,C 180,E1 -644.206,E2 -644.206} C_VEL
LIN {X 0,Y 601.432,Z 118.567,A -85,B 0,C 180,E1 -646.986,E2 -646.986} C_VEL
LIN {X 0,Y 601.417,Z 118.572,A -85,B 0,C 180,E1 -649.898,E2 -649.898} C_VEL
LIN {X 0,Y 601.456,Z 131.883,A -85,B 0,C 180,E1 -652.281,E2 -652.281} C_VEL
LIN {X 0,Y 601.402,Z 146.592,A -85,B 0,C 180,E1 -654.879,E2 -654.879} C_VEL
LIN {X 0,Y 601.654,Z 151.948,A -85,B 0,C 180,E1 -654.96,E2 -654.96} C_VEL
LIN {X 0,Y 601.56,Z 253.13,A -85,B 0,C 180,E1 -656.187,E2 -656.187} C_VEL
LIN {X 0,Y 601.533,Z 266.376,A -85,B 0,C 180,E1 -656.487,E2 -656.487} C_VEL
LIN {X 0,Y 601.541,Z 279.196,A -85,B 0,C 180,E1 -656.919,E2 -656.919} C_VEL
LIN {X 0,Y 601.479,Z 291.693,A -85,B 0,C 180,E1 -657.497,E2 -657.497} C_VEL
LIN {X 0,Y 601.437,Z 302.671,A -85,B 0,C 180,E1 -658.151,E2 -658.151} C_VEL
LIN {X 0,Y 601.458,Z 313.631,A -85,B 0,C 180,E1 -658.968,E2 -658.968} C_VEL
LIN {X 0,Y 601.413,Z 322.442,A -85,B 0,C 180,E1 -659.779,E2 -659.779} C_VEL
LIN {X 0,Y 601.407,Z 331.047,A -85,B 0,C 180,E1 -660.748,E2 -660.748} C_VEL
LIN {X 0,Y 601.394,Z 338.118,A -85,B 0,C 180,E1 -661.728,E2 -661.728} C_VEL
LIN {X 0,Y 601.361,Z 343.825,A -85,B 0,C 180,E1 -662.707,E2 -662.707} C_VEL
LIN {X 0,Y 601.363,Z 348.078,A -85,B 0,C 180,E1 -663.619,E2 -663.619} C_VEL
LIN {X 0,Y 601.34,Z 352.681,A -85,B 0,C 180,E1 -664.937,E2 -664.937} C_VEL
LIN {X 0,Y 601.314,Z 355.554,A -85,B 0,C 180,E1 -666.25,E2 -666.25} C_VEL
LIN {X 0,Y 601.33,Z 356.82,A -85,B 0,C 180,E1 -667.427,E2 -667.427} C_VEL
LIN {X 0,Y 601.316,Z 356.91,A -85,B 0,C 180,E1 -668.458,E2 -668.458} C_VEL
LIN {X 0,Y 601.314,Z 356.025,A -85,B 0,C 180,E1 -669.522,E2 -669.522} C_VEL
LIN {X 0,Y 601.33,Z 353.395,A -85,B 0,C 180,E1 -670.882,E2 -670.882} C_VEL
LIN {X 0,Y 601.358,Z 349.269,A -85,B 0,C 180,E1 -672.177,E2 -672.177} C_VEL
LIN {X 0,Y 601.344,Z 344.035,A -85,B 0,C 180,E1 -673.344,E2 -673.344} C_VEL
LIN {X 0,Y 601.398,Z 337.059,A -85,B 0,C 180,E1 -674.521,E2 -674.521} C_VEL
LIN {X 0,Y 601.398,Z 329.934,A -85,B 0,C 180,E1 -675.48,E2 -675.48} C_VEL
LIN {X 0,Y 601.432,Z 321.285,A -85,B 0,C 180,E1 -676.428,E2 -676.428} C_VEL
LIN {X 0,Y 601.449,Z 311.001,A -85,B 0,C 180,E1 -677.334,E2 -677.334} C_VEL
LIN {X 0,Y 601.448,Z 299.822,A -85,B 0,C 180,E1 -678.125,E2 -678.125} C_VEL
LIN {X 0,Y 601.511,Z 288.69,A -85,B 0,C 180,E1 -678.746,E2 -678.746} C_VEL
LIN {X 0,Y 601.567,Z 276.574,A -85,B 0,C 180,E1 -679.27,E2 -679.27} C_VEL
LIN {X 0,Y 601.558,Z 263.208,A -85,B 0,C 180,E1 -679.69,E2 -679.69} C_VEL
LIN {X 0,Y 601.56,Z 249.906,A -85,B 0,C 180,E1 -679.952,E2 -679.952} C_VEL
LIN {X 0,Y 601.587,Z 147.869,A -85,B 0,C 180,E1 -681.18,E2 -681.18} C_VEL
LIN {X 0,Y 601.392,Z 146.47,A -85,B 0,C 180,E1 -681.233,E2 -681.233} C_VEL
LIN {X 0,Y 601.453,Z 132.309,A -85,B 0,C 180,E1 -683.734,E2 -683.734} C_VEL
LIN {X 0,Y 601.424,Z 118.566,A -85,B 0,C 180,E1 -686.211,E2 -686.211} C_VEL
LIN {X 0,Y 601.413,Z 118.57,A -85,B 0,C 180,E1 -689.058,E2 -689.058} C_VEL
LIN {X 0,Y 601.43,Z 118.572,A -85,B 0,C 180,E1 -691.374,E2 -691.374} C_VEL
LIN {X 0,Y 601.395,Z 118.571,A -85,B 0,C 180,E1 -693.636,E2 -693.636} C_VEL
LIN {X 0,Y 601.412,Z 118.566,A -85,B 0,C 180,E1 -695.858,E2 -695.858} C_VEL
LIN {X 0,Y 601.405,Z 118.572,A -85,B 0,C 180,E1 -698.761,E2 -698.761} C_VEL
LIN {X 0,Y 601.387,Z 118.569,A -85,B 0,C 180,E1 -701.608,E2 -701.608} C_VEL
LIN {X 0,Y 601.41,Z 118.569,A -85,B 0,C 180,E1 -704.409,E2 -704.409} C_VEL
LIN {X 0,Y 601.381,Z 118.572,A -85,B 0,C 180,E1 -707.171,E2 -707.171} C_VEL
LIN {X 0,Y 601.424,Z 118.564,A -85,B 0,C 180,E1 -709.905,E2 -709.905} C_VEL
LIN {X 0,Y 601.406,Z 118.574,A -85,B 0,C 180,E1 -712.615,E2 -712.615} C_VEL
LIN {X 0,Y 601.384,Z 118.568,A -85,B 0,C 180,E1 -715.308,E2 -715.308} C_VEL
LIN {X 0,Y 601.434,Z 118.567,A -85,B 0,C 180,E1 -717.991,E2 -717.991} C_VEL
LIN {X 0,Y 601.402,Z 118.569,A -85,B 0,C 180,E1 -720.67,E2 -720.67} C_VEL
LIN {X 0,Y 601.407,Z 118.567,A -85,B 0,C 180,E1 -722.68,E2 -722.68} C_VEL
LIN {X 0,Y 601.391,Z 118.569,A -85,B 0,C 180,E1 -725.365,E2 -725.365} C_VEL
LIN {X 0,Y 601.431,Z 118.571,A -85,B 0,C 180,E1 -728.061,E2 -728.061} C_VEL
LIN {X 0,Y 601.375,Z 118.569,A -85,B 0,C 180,E1 -730.985,E2 -730.985} C_VEL
LIN {X 0,Y 601.385,Z 118.574,A -85,B 0,C 180,E1 -733.517,E2 -733.517} C_VEL
LIN {X 0,Y 601.382,Z 118.57,A -85,B 0,C 180,E1 -736.289,E2 -736.289} C_VEL
LIN {X 0,Y 601.367,Z 118.573,A -85,B 0,C 180,E1 -739.101,E2 -739.101} C_VEL
LIN {X 0,Y 601.389,Z 118.574,A -85,B 0,C 180,E1 -741.24,E2 -741.24} C_VEL
LIN {X 0,Y 601.38,Z 118.569,A -85,B 0,C 180,E1 -744.279,E2 -744.279} C_VEL
LIN {X 0,Y 601.421,Z 118.571,A -85,B 0,C 180,E1 -747.113,E2 -747.113} C_VEL
LIN {X 0,Y 601.381,Z 118.575,A -85,B 0,C 180,E1 -749.396,E2 -749.396} C_VEL
LIN {X 0,Y 601.384,Z 118.57,A -85,B 0,C 180,E1 -751.728,E2 -751.728} C_VEL
LIN {X 0,Y 601.405,Z 118.566,A -85,B 0,C 180,E1 -754.12,E2 -754.12} C_VEL
LIN {X 0,Y 601.437,Z 118.564,A -85,B 0,C 180,E1 -757.381,E2 -757.381} C_VEL
LIN {X 0,Y 601.379,Z 118.569,A -85,B 0,C 180,E1 -759.998,E2 -759.998} C_VEL
LIN {X 0,Y 601.389,Z 118.578,A -85,B 0,C 180,E1 -762.673,E2 -762.673} C_VEL
LIN {X 0,Y 601.404,Z 118.566,A -85,B 0,C 180,E1 -765.479,E2 -765.479} C_VEL
LIN {X 0,Y 601.422,Z 118.573,A -85,B 0,C 180,E1 -768.408,E2 -768.408} C_VEL
LIN {X 0,Y 601.409,Z 118.568,A -85,B 0,C 180,E1 -770.873,E2 -770.873} C_VEL
LIN {X 0,Y 601.396,Z 118.567,A -85,B 0,C 180,E1 -773.416,E2 -773.416} C_VEL
LIN {X 0,Y 601.433,Z 118.57,A -85,B 0,C 180,E1 -776.065,E2 -776.065} C_VEL
LIN {X 0,Y 601.404,Z 118.566,A -85,B 0,C 180,E1 -779.057,E2 -779.057} C_VEL
LIN {X 0,Y 601.413,Z 118.566,A -85,B 0,C 180,E1 -781.372,E2 -781.372} C_VEL
LIN {X 0,Y 601.412,Z 118.572,A -85,B 0,C 180,E1 -784.134,E2 -784.134} C_VEL
LIN {X 0,Y 601.422,Z 118.647,A -85,B 0,C 180,E1 -786.749,E2 -786.749} C_VEL
LIN {X 0,Y 601.692,Z 123.714,A -85,B 0,C 180,E1 -787.452,E2 -787.452} C_VEL
LIN {X 0,Y 601.629,Z 144.076,A -85,B 0,C 180,E1 -790.198,E2 -790.198} C_VEL
LIN {X 0,Y 601.535,Z 165.35,A -85,B 0,C 180,E1 -793.017,E2 -793.017} C_VEL
LIN {X 0,Y 601.456,Z 186.624,A -85,B 0,C 180,E1 -795.795,E2 -795.795} C_VEL
LIN {X 0,Y 601.426,Z 194.518,A -85,B 0,C 180,E1 -796.817,E2 -796.817} C_VEL
LIN {X 0,Y 601.638,Z 207.628,A -85,B 0,C 180,E1 -796.983,E2 -796.983} C_VEL
LIN {X 0,Y 601.613,Z 302.924,A -85,B 0,C 180,E1 -798.139,E2 -798.139} C_VEL
LIN {X 0,Y 601.56,Z 316.203,A -85,B 0,C 180,E1 -798.437,E2 -798.437} C_VEL
LIN {X 0,Y 601.543,Z 328.63,A -85,B 0,C 180,E1 -798.853,E2 -798.853} C_VEL
LIN {X 0,Y 601.523,Z 340.625,A -85,B 0,C 180,E1 -799.396,E2 -799.396} C_VEL
LIN {X 0,Y 601.483,Z 352.193,A -85,B 0,C 180,E1 -800.075,E2 -800.075} C_VEL
LIN {X 0,Y 601.444,Z 362.59,A -85,B 0,C 180,E1 -800.839,E2 -800.839} C_VEL
LIN {X 0,Y 601.429,Z 371.108,A -85,B 0,C 180,E1 -801.6,E2 -801.6} C_VEL
LIN {X 0,Y 601.418,Z 378.957,A -85,B 0,C 180,E1 -802.445,E2 -802.445} C_VEL
LIN {X 0,Y 601.37,Z 386.223,A -85,B 0,C 180,E1 -803.398,E2 -803.398} C_VEL
LIN {X 0,Y 601.372,Z 391.864,A -85,B 0,C 180,E1 -804.299,E2 -804.299} C_VEL
LIN {X 0,Y 601.336,Z 396.948,A -85,B 0,C 180,E1 -805.307,E2 -805.307} C_VEL
LIN {X 0,Y 601.368,Z 400.895,A -85,B 0,C 180,E1 -806.314,E2 -806.314} C_VEL
LIN {X 0,Y 601.325,Z 403.808,A -85,B 0,C 180,E1 -807.32,E2 -807.32} C_VEL
LIN {X 0,Y 601.343,Z 405.201,A -85,B 0,C 180,E1 -807.99,E2 -807.99} C_VEL
LIN {X 0,Y 601.339,Z 406.784,A -85,B 0,C 180,E1 -809.33,E2 -809.33} C_VEL
LIN {X 0,Y 601.335,Z 407,A -85,B 0,C 180,E1 -810,E2 -810} C_VEL
LIN {X 0,Y 601.347,Z 406.185,A -85,B 0,C 180,E1 -811.339,E2 -811.339} C_VEL
LIN {X 0,Y 601.343,Z 405.203,A -85,B 0,C 180,E1 -812.009,E2 -812.009} C_VEL
LIN {X 0,Y 601.325,Z 403.81,A -85,B 0,C 180,E1 -812.679,E2 -812.679} C_VEL
LIN {X 0,Y 601.368,Z 400.897,A -85,B 0,C 180,E1 -813.685,E2 -813.685} C_VEL
LIN {X 0,Y 601.336,Z 396.951,A -85,B 0,C 180,E1 -814.692,E2 -814.692} C_VEL
LIN {X 0,Y 601.373,Z 390.879,A -85,B 0,C 180,E1 -815.869,E2 -815.869} C_VEL
LIN {X 0,Y 601.381,Z 384.239,A -85,B 0,C 180,E1 -816.879,E2 -816.879} C_VEL
LIN {X 0,Y 601.4,Z 375.993,A -85,B 0,C 180,E1 -817.892,E2 -817.892} C_VEL
LIN {X 0,Y 601.436,Z 367.541,A -85,B 0,C 180,E1 -818.737,E2 -818.737} C_VEL
LIN {X 0,Y 601.449,Z 357.098,A -85,B 0,C 180,E1 -819.585,E2 -819.585} C_VEL
LIN {X 0,Y 601.467,Z 346.764,A -85,B 0,C 180,E1 -820.264,E2 -820.264} C_VEL
LIN {X 0,Y 601.537,Z 334.602,A -85,B 0,C 180,E1 -820.896,E2 -820.896} C_VEL
LIN {X 0,Y 601.554,Z 322.228,A -85,B 0,C 180,E1 -821.378,E2 -821.378} C_VEL
LIN {X 0,Y 601.583,Z 309.453,A -85,B 0,C 180,E1 -821.732,E2 -821.732} C_VEL
LIN {X 0,Y 601.623,Z 297.113,A -85,B 0,C 180,E1 -821.945,E2 -821.945} C_VEL
LIN {X 0,Y 601.504,Z 195.174,A -85,B 0,C 180,E1 -823.169,E2 -823.169} C_VEL
LIN {X 0,Y 601.444,Z 194.275,A -85,B 0,C 180,E1 -823.214,E2 -823.214} C_VEL
LIN {X 0,Y 601.516,Z 172.004,A -85,B 0,C 180,E1 -826.11,E2 -826.11} C_VEL
LIN {X 0,Y 601.531,Z 152.093,A -85,B 0,C 180,E1 -828.737,E2 -828.737} C_VEL
LIN {X 0,Y 601.655,Z 132.116,A -85,B 0,C 180,E1 -831.409,E2 -831.409} C_VEL
LIN {X 0,Y 601.673,Z 120.149,A -85,B 0,C 180,E1 -833.035,E2 -833.035} C_VEL
LIN {X 0,Y 601.409,Z 118.569,A -85,B 0,C 180,E1 -833.274,E2 -833.274} C_VEL
LIN {X 0,Y 601.413,Z 118.571,A -85,B 0,C 180,E1 -835.867,E2 -835.867} C_VEL
LIN {X 0,Y 601.401,Z 118.572,A -85,B 0,C 180,E1 -837.868,E2 -837.868} C_VEL
LIN {X 0,Y 601.43,Z 118.571,A -85,B 0,C 180,E1 -840.164,E2 -840.164} C_VEL
LIN {X 0,Y 601.412,Z 118.565,A -85,B 0,C 180,E1 -842.714,E2 -842.714} C_VEL
LIN {X 0,Y 601.389,Z 118.568,A -85,B 0,C 180,E1 -845.111,E2 -845.111} C_VEL
LIN {X 0,Y 601.436,Z 118.564,A -85,B 0,C 180,E1 -847.419,E2 -847.419} C_VEL
LIN {X 0,Y 601.412,Z 118.573,A -85,B 0,C 180,E1 -849.995,E2 -849.995} C_VEL
LIN {X 0,Y 601.407,Z 118.565,A -85,B 0,C 180,E1 -852.67,E2 -852.67} C_VEL
LIN {X 0,Y 601.427,Z 118.568,A -85,B 0,C 180,E1 -855.482,E2 -855.482} C_VEL
LIN {X 0,Y 601.42,Z 118.564,A -85,B 0,C 180,E1 -858.407,E2 -858.407} C_VEL
LIN {X 0,Y 601.43,Z 118.571,A -85,B 0,C 180,E1 -861.529,E2 -861.529} C_VEL
LIN {X 0,Y 601.382,Z 118.569,A -85,B 0,C 180,E1 -864.245,E2 -864.245} C_VEL
LIN {X 0,Y 601.417,Z 118.564,A -85,B 0,C 180,E1 -866.685,E2 -866.685} C_VEL
LIN {X 0,Y 601.412,Z 118.568,A -85,B 0,C 180,E1 -869.057,E2 -869.057} C_VEL
LIN {X 0,Y 601.431,Z 118.572,A -85,B 0,C 180,E1 -871.373,E2 -871.373} C_VEL
LIN {X 0,Y 601.399,Z 118.572,A -85,B 0,C 180,E1 -873.636,E2 -873.636} C_VEL
LIN {X 0,Y 601.417,Z 118.565,A -85,B 0,C 180,E1 -876.589,E2 -876.589} C_VEL
LIN {X 0,Y 601.426,Z 118.569,A -85,B 0,C 180,E1 -879.478,E2 -879.478} C_VEL
LIN {X 0,Y 601.392,Z 118.567,A -85,B 0,C 180,E1 -882.311,E2 -882.311} C_VEL
LIN {X 0,Y 601.411,Z 118.565,A -85,B 0,C 180,E1 -884.408,E2 -884.408} C_VEL
LIN {X 0,Y 601.412,Z 118.574,A -85,B 0,C 180,E1 -887.171,E2 -887.171} C_VEL
LIN {X 0,Y 601.434,Z 118.562,A -85,B 0,C 180,E1 -889.905,E2 -889.905} C_VEL
LIN {X 0,Y 601.442,Z 118.565,A -85,B 0,C 180,E1 -892.615,E2 -892.615} C_VEL
LIN {X 0,Y 601.411,Z 118.569,A -85,B 0,C 180,E1 -895.308,E2 -895.308} C_VEL
LIN {X 0,Y 601.437,Z 118.561,A -85,B 0,C 180,E1 -897.991,E2 -897.991} C_VEL
LIN {X 0,Y 601.454,Z 118.567,A -85,B 0,C 180,E1 -900.669,E2 -900.669} C_VEL
LIN {X 0,Y 601.419,Z 118.566,A -85,B 0,C 180,E1 -903.349,E2 -903.349} C_VEL
LIN {X 0,Y 601.442,Z 118.562,A -85,B 0,C 180,E1 -906.036,E2 -906.036} C_VEL
LIN {X 0,Y 601.436,Z 118.571,A -85,B 0,C 180,E1 -908.737,E2 -908.737} C_VEL
LIN {X 0,Y 601.42,Z 118.564,A -85,B 0,C 180,E1 -911.458,E2 -911.458} C_VEL
LIN {X 0,Y 601.41,Z 118.568,A -85,B 0,C 180,E1 -912.377,E2 -912.377} C_VEL
LIN {X 0,Y 600.743,Z 118.654,A -85,B 0,C 180,E1 -912.936,E2 -912.936} C_VEL
LIN {X 0,Y 597.892,Z 119.008,A -85,B 0,C 180,E1 -913.844,E2 -913.844} C_VEL
LIN {X 0,Y 595.481,Z 119.314,A -85,B 0,C 180,E1 -914.574,E2 -914.574} C_VEL
LIN {X 0,Y 594.443,Z 119.435,A -85,B 0,C 180,E1 -915.137,E2 -915.137} C_VEL
LIN {X 0,Y 594.357,Z 119.444,A -85,B 0,C 180,E1 -915.328,E2 -915.328} C_VEL
LIN {X 0,Y 594.386,Z 119.441,A -85,B 0,C 180,E1 -917.193,E2 -917.193} C_VEL
LIN {X 0,Y 594.373,Z 119.446,A -85,B 0,C 180,E1 -920.053,E2 -920.053} C_VEL
LIN {X 0,Y 594.36,Z 119.445,A -85,B 0,C 180,E1 -922.967,E2 -922.967} C_VEL
LIN {X 0,Y 594.374,Z 119.441,A -85,B 0,C 180,E1 -925.193,E2 -925.193} C_VEL
LIN {X 0,Y 594.382,Z 119.441,A -85,B 0,C 180,E1 -927.526,E2 -927.526} C_VEL
LIN {X 0,Y 594.384,Z 119.449,A -85,B 0,C 180,E1 -930.328,E2 -930.328} C_VEL
LIN {X 0,Y 594.375,Z 119.442,A -85,B 0,C 180,E1 -932.95,E2 -932.95} C_VEL
LIN {X 0,Y 594.351,Z 119.445,A -85,B 0,C 180,E1 -935.408,E2 -935.408} C_VEL
LIN {X 0,Y 594.386,Z 119.448,A -85,B 0,C 180,E1 -937.94,E2 -937.94} C_VEL
LIN {X 0,Y 594.378,Z 119.441,A -85,B 0,C 180,E1 -940.822,E2 -940.822} C_VEL
LIN {X 0,Y 594.379,Z 119.449,A -85,B 0,C 180,E1 -943.841,E2 -943.841} C_VEL
LIN {X 0,Y 594.376,Z 119.441,A -85,B 0,C 180,E1 -946.702,E2 -946.702} C_VEL
LIN {X 0,Y 594.371,Z 119.446,A -85,B 0,C 180,E1 -949.434,E2 -949.434} C_VEL
LIN {X 0,Y 594.388,Z 119.441,A -85,B 0,C 180,E1 -952.391,E2 -952.391} C_VEL
LIN {X 0,Y 594.35,Z 119.444,A -85,B 0,C 180,E1 -954.676,E2 -954.676} C_VEL
LIN {X 0,Y 594.376,Z 119.443,A -85,B 0,C 180,E1 -957.088,E2 -957.088} C_VEL
LIN {X 0,Y 594.383,Z 119.45,A -85,B 0,C 180,E1 -959.672,E2 -959.672} C_VEL
LIN {X 0,Y 594.37,Z 119.442,A -85,B 0,C 180,E1 -962.539,E2 -962.539} C_VEL
LIN {X 0,Y 594.372,Z 119.442,A -85,B 0,C 180,E1 -964.807,E2 -964.807} C_VEL
LIN {X 0,Y 594.361,Z 119.45,A -85,B 0,C 180,E1 -967.265,E2 -967.265} C_VEL
LIN {X 0,Y 594.372,Z 119.444,A -85,B 0,C 180,E1 -969.947,E2 -969.947} C_VEL
LIN {X 0,Y 594.387,Z 119.442,A -85,B 0,C 180,E1 -972.807,E2 -972.807} C_VEL
LIN {X 0,Y 594.385,Z 119.442,A -85,B 0,C 180,E1 -975.826,E2 -975.826} C_VEL
LIN {X 0,Y 594.39,Z 119.44,A -85,B 0,C 180,E1 -978.405,E2 -978.405} C_VEL
LIN {X 0,Y 594.394,Z 119.449,A -85,B 0,C 180,E1 -981.158,E2 -981.158} C_VEL
LIN {X 0,Y 594.394,Z 119.439,A -85,B 0,C 180,E1 -983.892,E2 -983.892} C_VEL
LIN {X 0,Y 594.377,Z 119.444,A -85,B 0,C 180,E1 -986.611,E2 -986.611} C_VEL
LIN {X 0,Y 594.417,Z 119.441,A -85,B 0,C 180,E1 -989.323,E2 -989.323} C_VEL
LIN {X 0,Y 594.406,Z 119.437,A -85,B 0,C 180,E1 -992.033,E2 -992.033} C_VEL
LIN {X 0,Y 594.387,Z 119.447,A -85,B 0,C 180,E1 -994.748,E2 -994.748} C_VEL
LIN {X 0,Y 594.391,Z 119.441,A -85,B 0,C 180,E1 -997.474,E2 -997.474} C_VEL
LIN {X 0,Y 594.396,Z 119.44,A -85,B 0,C 180,E1 -1000.216,E2 -1000.216} C_VEL
LIN {X 0,Y 594.364,Z 119.449,A -85,B 0,C 180,E1 -1002.984,E2 -1002.984} C_VEL
LIN {X 0,Y 594.37,Z 119.446,A -85,B 0,C 180,E1 -1005.078,E2 -1005.078} C_VEL
LIN {X 0,Y 594.388,Z 119.442,A -85,B 0,C 180,E1 -1007.194,E2 -1007.194} C_VEL
LIN {X 0,Y 594.397,Z 119.527,A -85,B 0,C 180,E1 -1009.851,E2 -1009.851} C_VEL
LIN {X 0,Y 594.419,Z 132.674,A -85,B 0,C 180,E1 -1012.232,E2 -1012.232} C_VEL
LIN {X 0,Y 594.349,Z 146.679,A -85,B 0,C 180,E1 -1014.732,E2 -1014.732} C_VEL
LIN {X 0,Y 594.758,Z 150.492,A -85,B 0,C 180,E1 -1014.788,E2 -1014.788} C_VEL
LIN {X 0,Y 594.617,Z 253.412,A -85,B 0,C 180,E1 -1016.052,E2 -1016.052} C_VEL
LIN {X 0,Y 594.596,Z 266.524,A -85,B 0,C 180,E1 -1016.354,E2 -1016.354} C_VEL
LIN {X 0,Y 594.567,Z 279.164,A -85,B 0,C 180,E1 -1016.786,E2 -1016.786} C_VEL
LIN {X 0,Y 594.484,Z 291.484,A -85,B 0,C 180,E1 -1017.361,E2 -1017.361} C_VEL
LIN {X 0,Y 594.428,Z 302.706,A -85,B 0,C 180,E1 -1018.036,E2 -1018.036} C_VEL
LIN {X 0,Y 594.421,Z 312.749,A -85,B 0,C 180,E1 -1018.787,E2 -1018.787} C_VEL
LIN {X 0,Y 594.377,Z 321.487,A -85,B 0,C 180,E1 -1019.582,E2 -1019.582} C_VEL
LIN {X 0,Y 594.322,Z 330.273,A -85,B 0,C 180,E1 -1020.563,E2 -1020.563} C_VEL
LIN {X 0,Y 594.325,Z 338.005,A -85,B 0,C 180,E1 -1021.635,E2 -1021.635} C_VEL
LIN {X 0,Y 594.268,Z 343.187,A -85,B 0,C 180,E1 -1022.523,E2 -1022.523} C_VEL
LIN {X 0,Y 594.267,Z 348.917,A -85,B 0,C 180,E1 -1023.769,E2 -1023.769} C_VEL
LIN {X 0,Y 594.254,Z 351.751,A -85,B 0,C 180,E1 -1024.589,E2 -1024.589} C_VEL
LIN {X 0,Y 594.224,Z 354.001,A -85,B 0,C 180,E1 -1025.418,E2 -1025.418} C_VEL
LIN {X 0,Y 594.221,Z 355.919,A -85,B 0,C 180,E1 -1026.463,E2 -1026.463} C_VEL
LIN {X 0,Y 594.227,Z 356.901,A -85,B 0,C 180,E1 -1027.589,E2 -1027.589} C_VEL
LIN {X 0,Y 594.207,Z 356.718,A -85,B 0,C 180,E1 -1028.819,E2 -1028.819} C_VEL
LIN {X 0,Y 594.227,Z 355.722,A -85,B 0,C 180,E1 -1029.758,E2 -1029.758} C_VEL
LIN {X 0,Y 594.23,Z 353.682,A -85,B 0,C 180,E1 -1030.806,E2 -1030.806} C_VEL
LIN {X 0,Y 594.262,Z 349.777,A -85,B 0,C 180,E1 -1032.086,E2 -1032.086} C_VEL
LIN {X 0,Y 594.275,Z 344.536,A -85,B 0,C 180,E1 -1033.308,E2 -1033.308} C_VEL
LIN {X 0,Y 594.308,Z 339.337,A -85,B 0,C 180,E1 -1034.244,E2 -1034.244} C_VEL
LIN {X 0,Y 594.32,Z 331.786,A -85,B 0,C 180,E1 -1035.336,E2 -1035.336} C_VEL
LIN {X 0,Y 594.345,Z 323.507,A -85,B 0,C 180,E1 -1036.298,E2 -1036.298} C_VEL
LIN {X 0,Y 594.385,Z 313.637,A -85,B 0,C 180,E1 -1037.231,E2 -1037.231} C_VEL
LIN {X 0,Y 594.431,Z 303.531,A -85,B 0,C 180,E1 -1037.999,E2 -1037.999} C_VEL
LIN {X 0,Y 594.503,Z 291.717,A -85,B 0,C 180,E1 -1038.716,E2 -1038.716} C_VEL
LIN {X 0,Y 594.582,Z 279.97,A -85,B 0,C 180,E1 -1039.272,E2 -1039.272} C_VEL
LIN {X 0,Y 594.596,Z 267.11,A -85,B 0,C 180,E1 -1039.719,E2 -1039.719} C_VEL
LIN {X 0,Y 594.618,Z 253.894,A -85,B 0,C 180,E1 -1040.029,E2 -1040.029} C_VEL
LIN {X 0,Y 594.757,Z 188.255,A -85,B 0,C 180,E1 -1040.844,E2 -1040.844} C_VEL
LIN {X 0,Y 594.707,Z 148.813,A -85,B 0,C 180,E1 -1041.324,E2 -1041.324} C_VEL
LIN {X 0,Y 594.348,Z 146.564,A -85,B 0,C 180,E1 -1041.375,E2 -1041.375} C_VEL
LIN {X 0,Y 594.428,Z 132.046,A -85,B 0,C 180,E1 -1043.971,E2 -1043.971} C_VEL
LIN {X 0,Y 594.378,Z 119.444,A -85,B 0,C 180,E1 -1046.265,E2 -1046.265} C_VEL
LIN {X 0,Y 594.37,Z 119.444,A -85,B 0,C 180,E1 -1048.65,E2 -1048.65} C_VEL
LIN {X 0,Y 594.385,Z 119.446,A -85,B 0,C 180,E1 -1051.043,E2 -1051.043} C_VEL
LIN {X 0,Y 594.378,Z 119.442,A -85,B 0,C 180,E1 -1053.98,E2 -1053.98} C_VEL
LIN {X 0,Y 594.358,Z 119.444,A -85,B 0,C 180,E1 -1056.295,E2 -1056.295} C_VEL
LIN {X 0,Y 594.394,Z 119.446,A -85,B 0,C 180,E1 -1059.225,E2 -1059.225} C_VEL
LIN {X 0,Y 594.34,Z 119.446,A -85,B 0,C 180,E1 -1062.095,E2 -1062.095} C_VEL
LIN {X 0,Y 594.359,Z 119.445,A -85,B 0,C 180,E1 -1064.219,E2 -1064.219} C_VEL
LIN {X 0,Y 594.373,Z 119.446,A -85,B 0,C 180,E1 -1066.321,E2 -1066.321} C_VEL
LIN {X 0,Y 594.354,Z 119.447,A -85,B 0,C 180,E1 -1069.095,E2 -1069.095} C_VEL
LIN {X 0,Y 594.376,Z 119.443,A -85,B 0,C 180,E1 -1071.843,E2 -1071.843} C_VEL
LIN {X 0,Y 594.38,Z 119.449,A -85,B 0,C 180,E1 -1074.573,E2 -1074.573} C_VEL
LIN {X 0,Y 594.372,Z 119.442,A -85,B 0,C 180,E1 -1077.289,E2 -1077.289} C_VEL
LIN {X 0,Y 594.415,Z 119.442,A -85,B 0,C 180,E1 -1080,E2 -1080} C_VEL
LIN {X 0,Y 594.375,Z 119.443,A -85,B 0,C 180,E1 -1082.711,E2 -1082.711} C_VEL
LIN {X 0,Y 594.361,Z 119.445,A -85,B 0,C 180,E1 -1085.428,E2 -1085.428} C_VEL
LIN {X 0,Y 594.373,Z 119.448,A -85,B 0,C 180,E1 -1088.158,E2 -1088.158} C_VEL
LIN {X 0,Y 594.336,Z 119.446,A -85,B 0,C 180,E1 -1091.044,E2 -1091.044} C_VEL
LIN {X 0,Y 594.35,Z 119.454,A -85,B 0,C 180,E1 -1093.68,E2 -1093.68} C_VEL
LIN {X 0,Y 594.313,Z 119.449,A -85,B 0,C 180,E1 -1096.691,E2 -1096.691} C_VEL
LIN {X 0,Y 594.334,Z 119.453,A -85,B 0,C 180,E1 -1099.336,E2 -1099.336} C_VEL
LIN {X 0,Y 594.344,Z 119.455,A -85,B 0,C 180,E1 -1101.504,E2 -1101.504} C_VEL
LIN {X 0,Y 594.344,Z 119.445,A -85,B 0,C 180,E1 -1104.448,E2 -1104.448} C_VEL
LIN {X 0,Y 594.358,Z 119.446,A -85,B 0,C 180,E1 -1106.701,E2 -1106.701} C_VEL
LIN {X 0,Y 594.337,Z 119.448,A -85,B 0,C 180,E1 -1109.779,E2 -1109.779} C_VEL
LIN {X 0,Y 594.343,Z 119.445,A -85,B 0,C 180,E1 -1112.149,E2 -1112.149} C_VEL
LIN {X 0,Y 594.368,Z 119.446,A -85,B 0,C 180,E1 -1114.581,E2 -1114.581} C_VEL
LIN {X 0,Y 594.385,Z 119.441,A -85,B 0,C 180,E1 -1117.607,E2 -1117.607} C_VEL
LIN {X 0,Y 594.362,Z 119.45,A -85,B 0,C 180,E1 -1120.568,E2 -1120.568} C_VEL
LIN {X 0,Y 594.349,Z 119.446,A -85,B 0,C 180,E1 -1123.301,E2 -1123.301} C_VEL
LIN {X 0,Y 594.349,Z 119.449,A -85,B 0,C 180,E1 -1126.163,E2 -1126.163} C_VEL
LIN {X 0,Y 594.377,Z 119.442,A -85,B 0,C 180,E1 -1129.179,E2 -1129.179} C_VEL
LIN {X 0,Y 594.376,Z 119.447,A -85,B 0,C 180,E1 -1132.058,E2 -1132.058} C_VEL
LIN {X 0,Y 594.352,Z 119.448,A -85,B 0,C 180,E1 -1134.677,E2 -1134.677} C_VEL
LIN {X 0,Y 594.378,Z 119.442,A -85,B 0,C 180,E1 -1137.089,E2 -1137.089} C_VEL
LIN {X 0,Y 594.374,Z 119.446,A -85,B 0,C 180,E1 -1139.675,E2 -1139.675} C_VEL
LIN {X 0,Y 594.38,Z 119.443,A -85,B 0,C 180,E1 -1142.539,E2 -1142.539} C_VEL
LIN {X 0,Y 594.403,Z 119.444,A -85,B 0,C 180,E1 -1145.564,E2 -1145.564} C_VEL
LIN {X 0,Y 594.391,Z 119.456,A -85,B 0,C 180,E1 -1146.573,E2 -1146.573} C_VEL
LIN {X 0,Y 594.792,Z 123.655,A -85,B 0,C 180,E1 -1147.168,E2 -1147.168} C_VEL
LIN {X 0,Y 594.673,Z 142.747,A -85,B 0,C 180,E1 -1149.776,E2 -1149.776} C_VEL
LIN {X 0,Y 594.575,Z 164.02,A -85,B 0,C 180,E1 -1152.634,E2 -1152.634} C_VEL
LIN {X 0,Y 594.45,Z 183.965,A -85,B 0,C 180,E1 -1155.274,E2 -1155.274} C_VEL
LIN {X 0,Y 594.434,Z 194.435,A -85,B 0,C 180,E1 -1156.648,E2 -1156.648} C_VEL
LIN {X 0,Y 594.75,Z 200.473,A -85,B 0,C 180,E1 -1156.743,E2 -1156.743} C_VEL
LIN {X 0,Y 594.666,Z 302.924,A -85,B 0,C 180,E1 -1157.999,E2 -1157.999} C_VEL
LIN {X 0,Y 594.602,Z 316.204,A -85,B 0,C 180,E1 -1158.3,E2 -1158.3} C_VEL
LIN {X 0,Y 594.599,Z 328.423,A -85,B 0,C 180,E1 -1158.713,E2 -1158.713} C_VEL
LIN {X 0,Y 594.536,Z 340.624,A -85,B 0,C 180,E1 -1159.27,E2 -1159.27} C_VEL
LIN {X 0,Y 594.477,Z 352.195,A -85,B 0,C 180,E1 -1159.957,E2 -1159.957} C_VEL
LIN {X 0,Y 594.414,Z 362.592,A -85,B 0,C 180,E1 -1160.729,E2 -1160.729} C_VEL
LIN {X 0,Y 594.383,Z 371.108,A -85,B 0,C 180,E1 -1161.5,E2 -1161.5} C_VEL
LIN {X 0,Y 594.347,Z 378.957,A -85,B 0,C 180,E1 -1162.355,E2 -1162.355} C_VEL
LIN {X 0,Y 594.283,Z 386.812,A -85,B 0,C 180,E1 -1163.408,E2 -1163.408} C_VEL
LIN {X 0,Y 594.289,Z 393.678,A -85,B 0,C 180,E1 -1164.571,E2 -1164.571} C_VEL
LIN {X 0,Y 594.27,Z 398.37,A -85,B 0,C 180,E1 -1165.591,E2 -1165.591} C_VEL
LIN {X 0,Y 594.267,Z 401.955,A -85,B 0,C 180,E1 -1166.61,E2 -1166.61} C_VEL
LIN {X 0,Y 594.226,Z 403.808,A -85,B 0,C 180,E1 -1167.288,E2 -1167.288} C_VEL
LIN {X 0,Y 594.242,Z 405.2,A -85,B 0,C 180,E1 -1167.966,E2 -1167.966} C_VEL
LIN {X 0,Y 594.239,Z 406.784,A -85,B 0,C 180,E1 -1169.322,E2 -1169.322} C_VEL
LIN {X 0,Y 594.236,Z 407,A -85,B 0,C 180,E1 -1170,E2 -1170} C_VEL
LIN {X 0,Y 594.247,Z 406.186,A -85,B 0,C 180,E1 -1171.355,E2 -1171.355} C_VEL
LIN {X 0,Y 594.242,Z 405.202,A -85,B 0,C 180,E1 -1172.033,E2 -1172.033} C_VEL
LIN {X 0,Y 594.226,Z 403.811,A -85,B 0,C 180,E1 -1172.711,E2 -1172.711} C_VEL
LIN {X 0,Y 594.289,Z 400.897,A -85,B 0,C 180,E1 -1173.729,E2 -1173.729} C_VEL
LIN {X 0,Y 594.241,Z 396.951,A -85,B 0,C 180,E1 -1174.748,E2 -1174.748} C_VEL
LIN {X 0,Y 594.305,Z 390.88,A -85,B 0,C 180,E1 -1175.939,E2 -1175.939} C_VEL
LIN {X 0,Y 594.308,Z 384.239,A -85,B 0,C 180,E1 -1176.962,E2 -1176.962} C_VEL
LIN {X 0,Y 594.359,Z 375.993,A -85,B 0,C 180,E1 -1177.986,E2 -1177.986} C_VEL
LIN {X 0,Y 594.382,Z 367.542,A -85,B 0,C 180,E1 -1178.842,E2 -1178.842} C_VEL
LIN {X 0,Y 594.432,Z 357.1,A -85,B 0,C 180,E1 -1179.699,E2 -1179.699} C_VEL
LIN {X 0,Y 594.481,Z 346.764,A -85,B 0,C 180,E1 -1180.386,E2 -1180.386} C_VEL
LIN {X 0,Y 594.558,Z 335.727,A -85,B 0,C 180,E1 -1180.973,E2 -1180.973} C_VEL
LIN {X 0,Y 594.579,Z 323.722,A -85,B 0,C 180,E1 -1181.464,E2 -1181.464} C_VEL
LIN {X 0,Y 594.647,Z 310.366,A -85,B 0,C 180,E1 -1181.85,E2 -1181.85} C_VEL
LIN {X 0,Y 594.697,Z 297.113,A -85,B 0,C 180,E1 -1182.087,E2 -1182.087} C_VEL
LIN {X 0,Y 594.621,Z 196.069,A -85,B 0,C 180,E1 -1183.314,E2 -1183.314} C_VEL
LIN {X 0,Y 594.434,Z 194.441,A -85,B 0,C 180,E1 -1183.351,E2 -1183.351} C_VEL
LIN {X 0,Y 594.536,Z 172.004,A -85,B 0,C 180,E1 -1186.304,E2 -1186.304} C_VEL
LIN {X 0,Y 594.583,Z 152.787,A -85,B 0,C 180,E1 -1188.87,E2 -1188.87} C_VEL
LIN {X 0,Y 594.768,Z 132.116,A -85,B 0,C 180,E1 -1191.67,E2 -1191.67} C_VEL
LIN {X 0,Y 594.754,Z 121.479,A -85,B 0,C 180,E1 -1193.135,E2 -1193.135} C_VEL
LIN {X 0,Y 594.376,Z 119.447,A -85,B 0,C 180,E1 -1193.45,E2 -1193.45} C_VEL
LIN {X 0,Y 594.386,Z 119.449,A -85,B 0,C 180,E1 -1196.022,E2 -1196.022} C_VEL
LIN {X 0,Y 594.376,Z 119.442,A -85,B 0,C 180,E1 -1198.998,E2 -1198.998} C_VEL
LIN {X 0,Y 594.377,Z 119.445,A -85,B 0,C 180,E1 -1201.642,E2 -1201.642} C_VEL
LIN {X 0,Y 594.375,Z 119.443,A -85,B 0,C 180,E1 -1204.58,E2 -1204.58} C_VEL
LIN {X 0,Y 594.39,Z 119.444,A -85,B 0,C 180,E1 -1207.608,E2 -1207.608} C_VEL
LIN {X 0,Y 594.364,Z 119.443,A -85,B 0,C 180,E1 -1210.567,E2 -1210.567} C_VEL
LIN {X 0,Y 594.366,Z 119.445,A -85,B 0,C 180,E1 -1213.299,E2 -1213.299} C_VEL
LIN {X 0,Y 594.368,Z 119.446,A -85,B 0,C 180,E1 -1216.16,E2 -1216.16} C_VEL
LIN {X 0,Y 594.378,Z 119.441,A -85,B 0,C 180,E1 -1218.536,E2 -1218.536} C_VEL
LIN {X 0,Y 594.382,Z 119.445,A -85,B 0,C 180,E1 -1221.295,E2 -1221.295} C_VEL
LIN {X 0,Y 594.35,Z 119.452,A -85,B 0,C 180,E1 -1223.755,E2 -1223.755} C_VEL
LIN {X 0,Y 594.364,Z 119.443,A -85,B 0,C 180,E1 -1226.237,E2 -1226.237} C_VEL
LIN {X 0,Y 594.369,Z 119.442,A -85,B 0,C 180,E1 -1228.649,E2 -1228.649} C_VEL
LIN {X 0,Y 594.383,Z 119.444,A -85,B 0,C 180,E1 -1231.042,E2 -1231.042} C_VEL
LIN {X 0,Y 594.381,Z 119.442,A -85,B 0,C 180,E1 -1233.978,E2 -1233.978} C_VEL
LIN {X 0,Y 594.384,Z 119.44,A -85,B 0,C 180,E1 -1236.295,E2 -1236.295} C_VEL
LIN {X 0,Y 594.403,Z 119.447,A -85,B 0,C 180,E1 -1239.224,E2 -1239.224} C_VEL
LIN {X 0,Y 594.344,Z 119.445,A -85,B 0,C 180,E1 -1242.094,E2 -1242.094} C_VEL
LIN {X 0,Y 594.363,Z 119.443,A -85,B 0,C 180,E1 -1244.219,E2 -1244.219} C_VEL
LIN {X 0,Y 594.382,Z 119.441,A -85,B 0,C 180,E1 -1246.321,E2 -1246.321} C_VEL
LIN {X 0,Y 594.373,Z 119.452,A -85,B 0,C 180,E1 -1249.094,E2 -1249.094} C_VEL
LIN {X 0,Y 594.41,Z 119.437,A -85,B 0,C 180,E1 -1251.843,E2 -1251.843} C_VEL
LIN {X 0,Y 594.399,Z 119.442,A -85,B 0,C 180,E1 -1254.572,E2 -1254.572} C_VEL
LIN {X 0,Y 594.399,Z 119.442,A -85,B 0,C 180,E1 -1257.289,E2 -1257.289} C_VEL
LIN {X 0,Y 594.414,Z 119.437,A -85,B 0,C 180,E1 -1260,E2 -1260} C_VEL
LIN {X 0,Y 594.407,Z 119.446,A -85,B 0,C 180,E1 -1262.71,E2 -1262.71} C_VEL
LIN {X 0,Y 594.389,Z 119.44,A -85,B 0,C 180,E1 -1265.427,E2 -1265.427} C_VEL
LIN {X 0,Y 594.417,Z 119.438,A -85,B 0,C 180,E1 -1268.156,E2 -1268.156} C_VEL
LIN {X 0,Y 594.389,Z 119.443,A -85,B 0,C 180,E1 -1271.074,E2 -1271.074} C_VEL
LIN {X 0,Y 594.377,Z 119.441,A -85,B 0,C 180,E1 -1273.679,E2 -1273.679} C_VEL
LIN {X 0,Y 594.357,Z 119.444,A -85,B 0,C 180,E1 -1275.328,E2 -1275.328} C_VEL
LIN {X 0,Y 593.683,Z 119.53,A -85,B 0,C 180,E1 -1275.894,E2 -1275.894} C_VEL
LIN {X 0,Y 590.818,Z 119.889,A -85,B 0,C 180,E1 -1276.812,E2 -1276.812} C_VEL
LIN {X 0,Y 588.408,Z 120.19,A -85,B 0,C 180,E1 -1277.551,E2 -1277.551} C_VEL
LIN {X 0,Y 587.385,Z 120.316,A -85,B 0,C 180,E1 -1278.121,E2 -1278.121} C_VEL
LIN {X 0,Y 587.309,Z 120.325,A -85,B 0,C 180,E1 -1278.314,E2 -1278.314} C_VEL
LIN {X 0,Y 587.327,Z 120.321,A -85,B 0,C 180,E1 -1281.037,E2 -1281.037} C_VEL
LIN {X 0,Y 587.319,Z 120.32,A -85,B 0,C 180,E1 -1283.258,E2 -1283.258} C_VEL
LIN {X 0,Y 587.333,Z 120.319,A -85,B 0,C 180,E1 -1285.516,E2 -1285.516} C_VEL
LIN {X 0,Y 587.345,Z 120.32,A -85,B 0,C 180,E1 -1287.817,E2 -1287.817} C_VEL
LIN {X 0,Y 587.339,Z 120.323,A -85,B 0,C 180,E1 -1290.511,E2 -1290.511} C_VEL
LIN {X 0,Y 587.336,Z 120.318,A -85,B 0,C 180,E1 -1293.112,E2 -1293.112} C_VEL
LIN {X 0,Y 587.343,Z 120.324,A -85,B 0,C 180,E1 -1295.896,E2 -1295.896} C_VEL
LIN {X 0,Y 587.331,Z 120.322,A -85,B 0,C 180,E1 -1298.479,E2 -1298.479} C_VEL
LIN {X 0,Y 587.334,Z 120.318,A -85,B 0,C 180,E1 -1301.156,E2 -1301.156} C_VEL
LIN {X 0,Y 587.33,Z 120.326,A -85,B 0,C 180,E1 -1304.114,E2 -1304.114} C_VEL
LIN {X 0,Y 587.318,Z 120.32,A -85,B 0,C 180,E1 -1306.994,E2 -1306.994} C_VEL
LIN {X 0,Y 587.317,Z 120.329,A -85,B 0,C 180,E1 -1309.746,E2 -1309.746} C_VEL
LIN {X 0,Y 587.343,Z 120.319,A -85,B 0,C 180,E1 -1312.393,E2 -1312.393} C_VEL
LIN {X 0,Y 587.322,Z 120.32,A -85,B 0,C 180,E1 -1314.944,E2 -1314.944} C_VEL
LIN {X 0,Y 587.338,Z 120.324,A -85,B 0,C 180,E1 -1317.421,E2 -1317.421} C_VEL
LIN {X 0,Y 587.33,Z 120.325,A -85,B 0,C 180,E1 -1319.83,E2 -1319.83} C_VEL
LIN {X 0,Y 587.348,Z 120.317,A -85,B 0,C 180,E1 -1322.307,E2 -1322.307} C_VEL
LIN {X 0,Y 587.332,Z 120.319,A -85,B 0,C 180,E1 -1324.484,E2 -1324.484} C_VEL
LIN {X 0,Y 587.337,Z 120.328,A -85,B 0,C 180,E1 -1327.486,E2 -1327.486} C_VEL
LIN {X 0,Y 587.34,Z 120.318,A -85,B 0,C 180,E1 -1330.425,E2 -1330.425} C_VEL
LIN {X 0,Y 587.348,Z 120.326,A -85,B 0,C 180,E1 -1333.311,E2 -1333.311} C_VEL
LIN {X 0,Y 587.356,Z 120.316,A -85,B 0,C 180,E1 -1336.155,E2 -1336.155} C_VEL
LIN {X 0,Y 587.341,Z 120.323,A -85,B 0,C 180,E1 -1338.963,E2 -1338.963} C_VEL
LIN {X 0,Y 587.367,Z 120.316,A -85,B 0,C 180,E1 -1341.745,E2 -1341.745} C_VEL
LIN {X 0,Y 587.361,Z 120.316,A -85,B 0,C 180,E1 -1344.507,E2 -1344.507} C_VEL
LIN {X 0,Y 587.37,Z 120.321,A -85,B 0,C 180,E1 -1347.257,E2 -1347.257} C_VEL
LIN {X 0,Y 587.382,Z 120.312,A -85,B 0,C 180,E1 -1350,E2 -1350} C_VEL
LIN {X 0,Y 587.37,Z 120.321,A -85,B 0,C 180,E1 -1352.744,E2 -1352.744} C_VEL
LIN {X 0,Y 587.362,Z 120.316,A -85,B 0,C 180,E1 -1355.493,E2 -1355.493} C_VEL
LIN {X 0,Y 587.368,Z 120.316,A -85,B 0,C 180,E1 -1358.256,E2 -1358.256} C_VEL
LIN {X 0,Y 587.346,Z 120.321,A -85,B 0,C 180,E1 -1361.134,E2 -1361.134} C_VEL
LIN {X 0,Y 587.363,Z 120.318,A -85,B 0,C 180,E1 -1364.261,E2 -1364.261} C_VEL
LIN {X 0,Y 587.349,Z 120.318,A -85,B 0,C 180,E1 -1367.406,E2 -1367.406} C_VEL
LIN {X 0,Y 587.346,Z 120.494,A -85,B 0,C 180,E1 -1369.803,E2 -1369.803} C_VEL
LIN {X 0,Y 587.405,Z 133.241,A -85,B 0,C 180,E1 -1372.141,E2 -1372.141} C_VEL
LIN {X 0,Y 587.308,Z 146.834,A -85,B 0,C 180,E1 -1374.572,E2 -1374.572} C_VEL
LIN {X 0,Y 587.854,Z 151.105,A -85,B 0,C 180,E1 -1374.637,E2 -1374.637} C_VEL
LIN {X 0,Y 587.682,Z 253.245,A -85,B 0,C 180,E1 -1375.905,E2 -1375.905} C_VEL
LIN {X 0,Y 587.649,Z 266.655,A -85,B 0,C 180,E1 -1376.218,E2 -1376.218} C_VEL
LIN {X 0,Y 587.584,Z 279.156,A -85,B 0,C 180,E1 -1376.65,E2 -1376.65} C_VEL
LIN {X 0,Y 587.504,Z 291.455,A -85,B 0,C 180,E1 -1377.231,E2 -1377.231} C_VEL
LIN {X 0,Y 587.413,Z 302.662,A -85,B 0,C 180,E1 -1377.912,E2 -1377.912} C_VEL
LIN {X 0,Y 587.405,Z 312.787,A -85,B 0,C 180,E1 -1378.678,E2 -1378.678} C_VEL
LIN {X 0,Y 587.327,Z 322.43,A -85,B 0,C 180,E1 -1379.578,E2 -1379.578} C_VEL
LIN {X 0,Y 587.272,Z 330.485,A -85,B 0,C 180,E1 -1380.5,E2 -1380.5} C_VEL
LIN {X 0,Y 587.241,Z 338.111,A -85,B 0,C 180,E1 -1381.574,E2 -1381.574} C_VEL
LIN {X 0,Y 587.173,Z 343.888,A -85,B 0,C 180,E1 -1382.59,E2 -1382.59} C_VEL
LIN {X 0,Y 587.168,Z 349.291,A -85,B 0,C 180,E1 -1383.82,E2 -1383.82} C_VEL
LIN {X 0,Y 587.128,Z 353.218,A -85,B 0,C 180,E1 -1385.07,E2 -1385.07} C_VEL
LIN {X 0,Y 587.125,Z 355.078,A -85,B 0,C 180,E1 -1385.912,E2 -1385.912} C_VEL
LIN {X 0,Y 587.123,Z 356.289,A -85,B 0,C 180,E1 -1386.764,E2 -1386.764} C_VEL
LIN {X 0,Y 587.119,Z 356.953,A -85,B 0,C 180,E1 -1387.811,E2 -1387.811} C_VEL
LIN {X 0,Y 587.113,Z 356.659,A -85,B 0,C 180,E1 -1388.916,E2 -1388.916} C_VEL
LIN {X 0,Y 587.143,Z 354.909,A -85,B 0,C 180,E1 -1390.269,E2 -1390.269} C_VEL
LIN {X 0,Y 587.166,Z 351.486,A -85,B 0,C 180,E1 -1391.629,E2 -1391.629} C_VEL
LIN {X 0,Y 587.18,Z 348.188,A -85,B 0,C 180,E1 -1392.552,E2 -1392.552} C_VEL
LIN {X 0,Y 587.182,Z 342.646,A -85,B 0,C 180,E1 -1393.736,E2 -1393.736} C_VEL
LIN {X 0,Y 587.22,Z 335.451,A -85,B 0,C 180,E1 -1394.921,E2 -1394.921} C_VEL
LIN {X 0,Y 587.266,Z 328.01,A -85,B 0,C 180,E1 -1395.893,E2 -1395.893} C_VEL
LIN {X 0,Y 587.347,Z 318.734,A -85,B 0,C 180,E1 -1396.879,E2 -1396.879} C_VEL
LIN {X 0,Y 587.422,Z 309.198,A -85,B 0,C 180,E1 -1397.703,E2 -1397.703} C_VEL
LIN {X 0,Y 587.44,Z 299.38,A -85,B 0,C 180,E1 -1398.396,E2 -1398.396} C_VEL
LIN {X 0,Y 587.518,Z 288.202,A -85,B 0,C 180,E1 -1399.028,E2 -1399.028} C_VEL
LIN {X 0,Y 587.601,Z 276.448,A -85,B 0,C 180,E1 -1399.545,E2 -1399.545} C_VEL
LIN {X 0,Y 587.65,Z 263.164,A -85,B 0,C 180,E1 -1399.971,E2 -1399.971} C_VEL
LIN {X 0,Y 587.71,Z 249.693,A -85,B 0,C 180,E1 -1400.24,E2 -1400.24} C_VEL
LIN {X 0,Y 587.82,Z 149.736,A -85,B 0,C 180,E1 -1401.471,E2 -1401.471} C_VEL
LIN {X 0,Y 587.314,Z 146.681,A -85,B 0,C 180,E1 -1401.52,E2 -1401.52} C_VEL
LIN {X 0,Y 587.435,Z 130.519,A -85,B 0,C 180,E1 -1404.444,E2 -1404.444} C_VEL
LIN {X 0,Y 587.344,Z 120.321,A -85,B 0,C 180,E1 -1406.347,E2 -1406.347} C_VEL
LIN {X 0,Y 587.326,Z 120.325,A -85,B 0,C 180,E1 -1409.034,E2 -1409.034} C_VEL
LIN {X 0,Y 587.323,Z 120.329,A -85,B 0,C 180,E1 -1411.403,E2 -1411.403} C_VEL
LIN {X 0,Y 587.339,Z 120.32,A -85,B 0,C 180,E1 -1413.824,E2 -1413.824} C_VEL
LIN {X 0,Y 587.298,Z 120.324,A -85,B 0,C 180,E1 -1415.992,E2 -1415.992} C_VEL
LIN {X 0,Y 587.335,Z 120.328,A -85,B 0,C 180,E1 -1418.963,E2 -1418.963} C_VEL
LIN {X 0,Y 587.342,Z 120.324,A -85,B 0,C 180,E1 -1421.151,E2 -1421.151} C_VEL
LIN {X 0,Y 587.311,Z 120.322,A -85,B 0,C 180,E1 -1424.025,E2 -1424.025} C_VEL
LIN {X 0,Y 587.351,Z 120.319,A -85,B 0,C 180,E1 -1426.154,E2 -1426.154} C_VEL
LIN {X 0,Y 587.342,Z 120.323,A -85,B 0,C 180,E1 -1428.963,E2 -1428.963} C_VEL
LIN {X 0,Y 587.336,Z 120.319,A -85,B 0,C 180,E1 -1431.745,E2 -1431.745} C_VEL
LIN {X 0,Y 587.346,Z 120.326,A -85,B 0,C 180,E1 -1434.507,E2 -1434.507} C_VEL
LIN {X 0,Y 587.341,Z 120.318,A -85,B 0,C 180,E1 -1437.257,E2 -1437.257} C_VEL
LIN {X 0,Y 587.383,Z 120.318,A -85,B 0,C 180,E1 -1440,E2 -1440} C_VEL
LIN {X 0,Y 587.342,Z 120.319,A -85,B 0,C 180,E1 -1442.744,E2 -1442.744} C_VEL
LIN {X 0,Y 587.33,Z 120.321,A -85,B 0,C 180,E1 -1445.494,E2 -1445.494} C_VEL
LIN {X 0,Y 587.329,Z 120.324,A -85,B 0,C 180,E1 -1448.256,E2 -1448.256} C_VEL
LIN {X 0,Y 587.302,Z 120.323,A -85,B 0,C 180,E1 -1451.107,E2 -1451.107} C_VEL
LIN {X 0,Y 587.322,Z 120.328,A -85,B 0,C 180,E1 -1453.847,E2 -1453.847} C_VEL
LIN {X 0,Y 587.274,Z 120.326,A -85,B 0,C 180,E1 -1456.788,E2 -1456.788} C_VEL
LIN {X 0,Y 587.283,Z 120.334,A -85,B 0,C 180,E1 -1459.577,E2 -1459.577} C_VEL
LIN {X 0,Y 587.274,Z 120.331,A -85,B 0,C 180,E1 -1461.777,E2 -1461.777} C_VEL
LIN {X 0,Y 587.29,Z 120.324,A -85,B 0,C 180,E1 -1464.565,E2 -1464.565} C_VEL
LIN {X 0,Y 587.305,Z 120.329,A -85,B 0,C 180,E1 -1467.048,E2 -1467.048} C_VEL
LIN {X 0,Y 587.297,Z 120.323,A -85,B 0,C 180,E1 -1470.173,E2 -1470.173} C_VEL
LIN {X 0,Y 587.335,Z 120.327,A -85,B 0,C 180,E1 -1473.11,E2 -1473.11} C_VEL
LIN {X 0,Y 587.28,Z 120.325,A -85,B 0,C 180,E1 -1475.901,E2 -1475.901} C_VEL
LIN {X 0,Y 587.316,Z 120.325,A -85,B 0,C 180,E1 -1478.481,E2 -1478.481} C_VEL
LIN {X 0,Y 587.334,Z 120.322,A -85,B 0,C 180,E1 -1481.157,E2 -1481.157} C_VEL
LIN {X 0,Y 587.307,Z 120.324,A -85,B 0,C 180,E1 -1484.111,E2 -1484.111} C_VEL
LIN {X 0,Y 587.293,Z 120.327,A -85,B 0,C 180,E1 -1486.991,E2 -1486.991} C_VEL
LIN {X 0,Y 587.309,Z 120.323,A -85,B 0,C 180,E1 -1489.745,E2 -1489.745} C_VEL
LIN {X 0,Y 587.344,Z 120.327,A -85,B 0,C 180,E1 -1492.392,E2 -1492.392} C_VEL
LIN {X 0,Y 587.357,Z 120.32,A -85,B 0,C 180,E1 -1495.779,E2 -1495.779} C_VEL
LIN {X 0,Y 587.336,Z 120.327,A -85,B 0,C 180,E1 -1498.23,E2 -1498.23} C_VEL
LIN {X 0,Y 587.348,Z 120.318,A -85,B 0,C 180,E1 -1500.868,E2 -1500.868} C_VEL
LIN {X 0,Y 587.312,Z 120.329,A -85,B 0,C 180,E1 -1503.72,E2 -1503.72} C_VEL
LIN {X 0,Y 587.365,Z 120.423,A -85,B 0,C 180,E1 -1506.463,E2 -1506.463} C_VEL
LIN {X 0,Y 587.881,Z 126.149,A -85,B 0,C 180,E1 -1507.259,E2 -1507.259} C_VEL
LIN {X 0,Y 587.744,Z 146.736,A -85,B 0,C 180,E1 -1510.074,E2 -1510.074} C_VEL
LIN {X 0,Y 587.57,Z 167.73,A -85,B 0,C 180,E1 -1512.921,E2 -1512.921} C_VEL
LIN {X 0,Y 587.438,Z 188.613,A -85,B 0,C 180,E1 -1515.713,E2 -1515.713} C_VEL
LIN {X 0,Y 587.402,Z 194.435,A -85,B 0,C 180,E1 -1516.486,E2 -1516.486} C_VEL
LIN {X 0,Y 587.841,Z 198.685,A -85,B 0,C 180,E1 -1516.562,E2 -1516.562} C_VEL
LIN {X 0,Y 587.726,Z 302.924,A -85,B 0,C 180,E1 -1517.855,E2 -1517.855} C_VEL
LIN {X 0,Y 587.668,Z 316.205,A -85,B 0,C 180,E1 -1518.16,E2 -1518.16} C_VEL
LIN {X 0,Y 587.629,Z 328.628,A -85,B 0,C 180,E1 -1518.585,E2 -1518.585} C_VEL
LIN {X 0,Y 587.558,Z 340.622,A -85,B 0,C 180,E1 -1519.141,E2 -1519.141} C_VEL
LIN {X 0,Y 587.464,Z 352.197,A -85,B 0,C 180,E1 -1519.836,E2 -1519.836} C_VEL
LIN {X 0,Y 587.366,Z 362.594,A -85,B 0,C 180,E1 -1520.617,E2 -1520.617} C_VEL
LIN {X 0,Y 587.322,Z 371.108,A -85,B 0,C 180,E1 -1521.397,E2 -1521.397} C_VEL
LIN {X 0,Y 587.274,Z 378.957,A -85,B 0,C 180,E1 -1522.262,E2 -1522.262} C_VEL
LIN {X 0,Y 587.231,Z 385.466,A -85,B 0,C 180,E1 -1523.126,E2 -1523.126} C_VEL
LIN {X 0,Y 587.237,Z 391.864,A -85,B 0,C 180,E1 -1524.161,E2 -1524.161} C_VEL
LIN {X 0,Y 587.147,Z 396.948,A -85,B 0,C 180,E1 -1525.193,E2 -1525.193} C_VEL
LIN {X 0,Y 587.213,Z 400.894,A -85,B 0,C 180,E1 -1526.225,E2 -1526.225} C_VEL
LIN {X 0,Y 587.132,Z 403.807,A -85,B 0,C 180,E1 -1527.255,E2 -1527.255} C_VEL
LIN {X 0,Y 587.141,Z 405.199,A -85,B 0,C 180,E1 -1527.942,E2 -1527.942} C_VEL
LIN {X 0,Y 587.14,Z 406.784,A -85,B 0,C 180,E1 -1529.314,E2 -1529.314} C_VEL
LIN {X 0,Y 587.137,Z 407,A -85,B 0,C 180,E1 -1530,E2 -1530} C_VEL
LIN {X 0,Y 587.147,Z 406.186,A -85,B 0,C 180,E1 -1531.371,E2 -1531.371} C_VEL
LIN {X 0,Y 587.141,Z 405.201,A -85,B 0,C 180,E1 -1532.058,E2 -1532.058} C_VEL
LIN {X 0,Y 587.132,Z 403.811,A -85,B 0,C 180,E1 -1532.744,E2 -1532.744} C_VEL
LIN {X 0,Y 587.213,Z 400.897,A -85,B 0,C 180,E1 -1533.774,E2 -1533.774} C_VEL
LIN {X 0,Y 587.147,Z 396.951,A -85,B 0,C 180,E1 -1534.806,E2 -1534.806} C_VEL
LIN {X 0,Y 587.218,Z 390.879,A -85,B 0,C 180,E1 -1536.011,E2 -1536.011} C_VEL
LIN {X 0,Y 587.245,Z 384.24,A -85,B 0,C 180,E1 -1537.046,E2 -1537.046} C_VEL
LIN {X 0,Y 587.299,Z 375.994,A -85,B 0,C 180,E1 -1538.083,E2 -1538.083} C_VEL
LIN {X 0,Y 587.343,Z 367.542,A -85,B 0,C 180,E1 -1538.949,E2 -1538.949} C_VEL
LIN {X 0,Y 587.419,Z 357.102,A -85,B 0,C 180,E1 -1539.816,E2 -1539.816} C_VEL
LIN {X 0,Y 587.497,Z 346.762,A -85,B 0,C 180,E1 -1540.511,E2 -1540.511} C_VEL
LIN {X 0,Y 587.56,Z 334.824,A -85,B 0,C 180,E1 -1541.148,E2 -1541.148} C_VEL
LIN {X 0,Y 587.629,Z 322.609,A -85,B 0,C 180,E1 -1541.639,E2 -1541.639} C_VEL
LIN {X 0,Y 587.703,Z 309.451,A -85,B 0,C 180,E1 -1542.014,E2 -1542.014} C_VEL
LIN {X 0,Y 587.776,Z 297.113,A -85,B 0,C 180,E1 -1542.231,E2 -1542.231} C_VEL
LIN {X 0,Y 587.714,Z 196.737,A -85,B 0,C 180,E1 -1543.465,E2 -1543.465} C_VEL
LIN {X 0,Y 587.401,Z 194.441,A -85,B 0,C 180,E1 -1543.514,E2 -1543.514} C_VEL
LIN {X 0,Y 587.556,Z 173.334,A -85,B 0,C 180,E1 -1546.325,E2 -1546.325} C_VEL
LIN {X 0,Y 587.668,Z 152.572,A -85,B 0,C 180,E1 -1549.13,E2 -1549.13} C_VEL
LIN {X 0,Y 587.873,Z 132.091,A -85,B 0,C 180,E1 -1551.937,E2 -1551.937} C_VEL
LIN {X 0,Y 587.751,Z 122.581,A -85,B 0,C 180,E1 -1553.24,E2 -1553.24} C_VEL
LIN {X 0,Y 587.342,Z 120.325,A -85,B 0,C 180,E1 -1553.584,E2 -1553.584} C_VEL
LIN {X 0,Y 587.339,Z 120.327,A -85,B 0,C 180,E1 -1556.278,E2 -1556.278} C_VEL
LIN {X 0,Y 587.346,Z 120.317,A -85,B 0,C 180,E1 -1559.132,E2 -1559.132} C_VEL
LIN {X 0,Y 587.342,Z 120.324,A -85,B 0,C 180,E1 -1561.835,E2 -1561.835} C_VEL
LIN {X 0,Y 587.345,Z 120.321,A -85,B 0,C 180,E1 -1564.347,E2 -1564.347} C_VEL
LIN {X 0,Y 587.345,Z 120.322,A -85,B 0,C 180,E1 -1567.607,E2 -1567.607} C_VEL
LIN {X 0,Y 587.316,Z 120.324,A -85,B 0,C 180,E1 -1570.254,E2 -1570.254} C_VEL
LIN {X 0,Y 587.314,Z 120.322,A -85,B 0,C 180,E1 -1573.118,E2 -1573.118} C_VEL
LIN {X 0,Y 587.323,Z 120.325,A -85,B 0,C 180,E1 -1576.049,E2 -1576.049} C_VEL
LIN {X 0,Y 587.336,Z 120.319,A -85,B 0,C 180,E1 -1578.925,E2 -1578.925} C_VEL
LIN {X 0,Y 587.328,Z 120.327,A -85,B 0,C 180,E1 -1581.52,E2 -1581.52} C_VEL
LIN {X 0,Y 587.29,Z 120.326,A -85,B 0,C 180,E1 -1584.099,E2 -1584.099} C_VEL
LIN {X 0,Y 587.337,Z 120.319,A -85,B 0,C 180,E1 -1586.888,E2 -1586.888} C_VEL
LIN {X 0,Y 587.326,Z 120.329,A -85,B 0,C 180,E1 -1589.491,E2 -1589.491} C_VEL
LIN {X 0,Y 587.351,Z 120.316,A -85,B 0,C 180,E1 -1592.307,E2 -1592.307} C_VEL
LIN {X 0,Y 587.35,Z 120.325,A -85,B 0,C 180,E1 -1595.241,E2 -1595.241} C_VEL
LIN {X 0,Y 587.32,Z 120.32,A -85,B 0,C 180,E1 -1598.225,E2 -1598.225} C_VEL
LIN {X 0,Y 587.347,Z 120.326,A -85,B 0,C 180,E1 -1601.151,E2 -1601.151} C_VEL
LIN {X 0,Y 587.32,Z 120.32,A -85,B 0,C 180,E1 -1604.024,E2 -1604.024} C_VEL
LIN {X 0,Y 587.359,Z 120.315,A -85,B 0,C 180,E1 -1606.154,E2 -1606.154} C_VEL
LIN {X 0,Y 587.339,Z 120.326,A -85,B 0,C 180,E1 -1608.962,E2 -1608.962} C_VEL
LIN {X 0,Y 587.362,Z 120.315,A -85,B 0,C 180,E1 -1611.744,E2 -1611.744} C_VEL
LIN {X 0,Y 587.365,Z 120.318,A -85,B 0,C 180,E1 -1614.507,E2 -1614.507} C_VEL
LIN {X 0,Y 587.366,Z 120.319,A -85,B 0,C 180,E1 -1617.256,E2 -1617.256} C_VEL
LIN {X 0,Y 587.383,Z 120.312,A -85,B 0,C 180,E1 -1620,E2 -1620} C_VEL
LIN {X 0,Y 587.373,Z 120.323,A -85,B 0,C 180,E1 -1622.743,E2 -1622.743} C_VEL
LIN {X 0,Y 587.357,Z 120.316,A -85,B 0,C 180,E1 -1625.493,E2 -1625.493} C_VEL
LIN {X 0,Y 587.37,Z 120.317,A -85,B 0,C 180,E1 -1628.255,E2 -1628.255} C_VEL
LIN {X 0,Y 587.346,Z 120.319,A -85,B 0,C 180,E1 -1631.133,E2 -1631.133} C_VEL
LIN {X 0,Y 587.363,Z 120.32,A -85,B 0,C 180,E1 -1634.26,E2 -1634.26} C_VEL
LIN {X 0,Y 587.347,Z 120.317,A -85,B 0,C 180,E1 -1637.406,E2 -1637.406} C_VEL
LIN {X 0,Y 587.309,Z 120.325,A -85,B 0,C 180,E1 -1638.314,E2 -1638.314} C_VEL
LIN {X 0,Y 586.665,Z 120.405,A -85,B 0,C 180,E1 -1638.886,E2 -1638.886} C_VEL
LIN {X 0,Y 583.839,Z 120.755,A -85,B 0,C 180,E1 -1639.815,E2 -1639.815} C_VEL
LIN {X 0,Y 581.428,Z 121.062,A -85,B 0,C 180,E1 -1640.562,E2 -1640.562} C_VEL
LIN {X 0,Y 580.375,Z 121.187,A -85,B 0,C 180,E1 -1641.138,E2 -1641.138} C_VEL
LIN {X 0,Y 580.28,Z 121.197,A -85,B 0,C 180,E1 -1641.333,E2 -1641.333} C_VEL
LIN {X 0,Y 580.298,Z 121.205,A -85,B 0,C 180,E1 -1644.316,E2 -1644.316} C_VEL
LIN {X 0,Y 580.303,Z 121.199,A -85,B 0,C 180,E1 -1646.622,E2 -1646.622} C_VEL
LIN {X 0,Y 580.298,Z 121.195,A -85,B 0,C 180,E1 -1649.31,E2 -1649.31} C_VEL
LIN {X 0,Y 580.299,Z 121.205,A -85,B 0,C 180,E1 -1652.2,E2 -1652.2} C_VEL
LIN {X 0,Y 580.286,Z 121.198,A -85,B 0,C 180,E1 -1654.696,E2 -1654.696} C_VEL
LIN {X 0,Y 580.297,Z 121.195,A -85,B 0,C 180,E1 -1657.268,E2 -1657.268} C_VEL
LIN {X 0,Y 580.295,Z 121.201,A -85,B 0,C 180,E1 -1660.271,E2 -1660.271} C_VEL
LIN {X 0,Y 580.277,Z 121.198,A -85,B 0,C 180,E1 -1662.706,E2 -1662.706} C_VEL
LIN {X 0,Y 580.27,Z 121.203,A -85,B 0,C 180,E1 -1665.608,E2 -1665.608} C_VEL
LIN {X 0,Y 580.31,Z 121.197,A -85,B 0,C 180,E1 -1668.234,E2 -1668.234} C_VEL
LIN {X 0,Y 580.287,Z 121.196,A -85,B 0,C 180,E1 -1670.966,E2 -1670.966} C_VEL
LIN {X 0,Y 580.279,Z 121.205,A -85,B 0,C 180,E1 -1673.598,E2 -1673.598} C_VEL
LIN {X 0,Y 580.312,Z 121.196,A -85,B 0,C 180,E1 -1676.145,E2 -1676.145} C_VEL
LIN {X 0,Y 580.285,Z 121.196,A -85,B 0,C 180,E1 -1678.615,E2 -1678.615} C_VEL
LIN {X 0,Y 580.291,Z 121.198,A -85,B 0,C 180,E1 -1681.024,E2 -1681.024} C_VEL
LIN {X 0,Y 580.288,Z 121.204,A -85,B 0,C 180,E1 -1683.666,E2 -1683.666} C_VEL
LIN {X 0,Y 580.296,Z 121.202,A -85,B 0,C 180,E1 -1685.684,E2 -1685.684} C_VEL
LIN {X 0,Y 580.271,Z 121.201,A -85,B 0,C 180,E1 -1687.948,E2 -1687.948} C_VEL
LIN {X 0,Y 580.315,Z 121.196,A -85,B 0,C 180,E1 -1690.914,E2 -1690.914} C_VEL
LIN {X 0,Y 580.276,Z 121.2,A -85,B 0,C 180,E1 -1693.826,E2 -1693.826} C_VEL
LIN {X 0,Y 580.322,Z 121.193,A -85,B 0,C 180,E1 -1695.983,E2 -1695.983} C_VEL
LIN {X 0,Y 580.301,Z 121.198,A -85,B 0,C 180,E1 -1698.827,E2 -1698.827} C_VEL
LIN {X 0,Y 580.331,Z 121.194,A -85,B 0,C 180,E1 -1701.644,E2 -1701.644} C_VEL
LIN {X 0,Y 580.329,Z 121.192,A -85,B 0,C 180,E1 -1704.441,E2 -1704.441} C_VEL
LIN {X 0,Y 580.344,Z 121.189,A -85,B 0,C 180,E1 -1707.918,E2 -1707.918} C_VEL
LIN {X 0,Y 580.359,Z 121.192,A -85,B 0,C 180,E1 -1710.694,E2 -1710.694} C_VEL
LIN {X 0,Y 580.281,Z 121.199,A -85,B 0,C 180,E1 -1713.472,E2 -1713.472} C_VEL
LIN {X 0,Y 580.329,Z 121.192,A -85,B 0,C 180,E1 -1715.56,E2 -1715.56} C_VEL
LIN {X 0,Y 580.331,Z 121.194,A -85,B 0,C 180,E1 -1718.356,E2 -1718.356} C_VEL
LIN {X 0,Y 580.298,Z 121.198,A -85,B 0,C 180,E1 -1721.192,E2 -1721.192} C_VEL
LIN {X 0,Y 580.324,Z 121.193,A -85,B 0,C 180,E1 -1724.017,E2 -1724.017} C_VEL
LIN {X 0,Y 580.31,Z 121.2,A -85,B 0,C 180,E1 -1726.914,E2 -1726.914} C_VEL
LIN {X 0,Y 580.321,Z 121.279,A -85,B 0,C 180,E1 -1729.721,E2 -1729.721} C_VEL
LIN {X 0,Y 580.396,Z 133.806,A -85,B 0,C 180,E1 -1732.048,E2 -1732.048} C_VEL
LIN {X 0,Y 580.265,Z 146.74,A -85,B 0,C 180,E1 -1734.404,E2 -1734.404} C_VEL
LIN {X 0,Y 580.972,Z 151.424,A -85,B 0,C 180,E1 -1734.479,E2 -1734.479} C_VEL
LIN {X 0,Y 580.753,Z 253.113,A -85,B 0,C 180,E1 -1735.755,E2 -1735.755} C_VEL
LIN {X 0,Y 580.705,Z 266.595,A -85,B 0,C 180,E1 -1736.072,E2 -1736.072} C_VEL
LIN {X 0,Y 580.611,Z 277.916,A -85,B 0,C 180,E1 -1736.462,E2 -1736.462} C_VEL
LIN {X 0,Y 580.547,Z 289.608,A -85,B 0,C 180,E1 -1736.999,E2 -1736.999} C_VEL
LIN {X 0,Y 580.452,Z 301.329,A -85,B 0,C 180,E1 -1737.698,E2 -1737.698} C_VEL
LIN {X 0,Y 580.36,Z 311.762,A -85,B 0,C 180,E1 -1738.478,E2 -1738.478} C_VEL
LIN {X 0,Y 580.289,Z 320.818,A -85,B 0,C 180,E1 -1739.308,E2 -1739.308} C_VEL
LIN {X 0,Y 580.217,Z 328.664,A -85,B 0,C 180,E1 -1740.178,E2 -1740.178} C_VEL
LIN {X 0,Y 580.151,Z 336.228,A -85,B 0,C 180,E1 -1741.201,E2 -1741.201} C_VEL
LIN {X 0,Y 580.143,Z 342.263,A -85,B 0,C 180,E1 -1742.211,E2 -1742.211} C_VEL
LIN {X 0,Y 580.087,Z 347.376,A -85,B 0,C 180,E1 -1743.285,E2 -1743.285} C_VEL
LIN {X 0,Y 580.073,Z 351.822,A -85,B 0,C 180,E1 -1744.527,E2 -1744.527} C_VEL
LIN {X 0,Y 580.028,Z 354.774,A -85,B 0,C 180,E1 -1745.727,E2 -1745.727} C_VEL
LIN {X 0,Y 580.031,Z 356.459,A -85,B 0,C 180,E1 -1746.9,E2 -1746.9} C_VEL
LIN {X 0,Y 580.015,Z 356.979,A -85,B 0,C 180,E1 -1748.168,E2 -1748.168} C_VEL
LIN {X 0,Y 580.019,Z 356.496,A -85,B 0,C 180,E1 -1749.152,E2 -1749.152} C_VEL
LIN {X 0,Y 580.043,Z 355.011,A -85,B 0,C 180,E1 -1750.242,E2 -1750.242} C_VEL
LIN {X 0,Y 580.042,Z 352.58,A -85,B 0,C 180,E1 -1751.305,E2 -1751.305} C_VEL
LIN {X 0,Y 580.092,Z 349.186,A -85,B 0,C 180,E1 -1752.351,E2 -1752.351} C_VEL
LIN {X 0,Y 580.108,Z 344.831,A -85,B 0,C 180,E1 -1753.374,E2 -1753.374} C_VEL
LIN {X 0,Y 580.155,Z 339.429,A -85,B 0,C 180,E1 -1754.38,E2 -1754.38} C_VEL
LIN {X 0,Y 580.183,Z 332.902,A -85,B 0,C 180,E1 -1755.366,E2 -1755.366} C_VEL
LIN {X 0,Y 580.228,Z 325.011,A -85,B 0,C 180,E1 -1756.338,E2 -1756.338} C_VEL
LIN {X 0,Y 580.315,Z 315.392,A -85,B 0,C 180,E1 -1757.298,E2 -1757.298} C_VEL
LIN {X 0,Y 580.415,Z 304.61,A -85,B 0,C 180,E1 -1758.167,E2 -1758.167} C_VEL
LIN {X 0,Y 580.455,Z 294.186,A -85,B 0,C 180,E1 -1758.839,E2 -1758.839} C_VEL
LIN {X 0,Y 580.611,Z 281.69,A -85,B 0,C 180,E1 -1759.469,E2 -1759.469} C_VEL
LIN {X 0,Y 580.699,Z 269.338,A -85,B 0,C 180,E1 -1759.936,E2 -1759.936} C_VEL
LIN {X 0,Y 580.744,Z 256.843,A -85,B 0,C 180,E1 -1760.262,E2 -1760.262} C_VEL
LIN {X 0,Y 580.801,Z 240.01,A -85,B 0,C 180,E1 -1760.514,E2 -1760.514} C_VEL
LIN {X 0,Y 580.884,Z 150.493,A -85,B 0,C 180,E1 -1761.625,E2 -1761.625} C_VEL
LIN {X 0,Y 580.254,Z 146.593,A -85,B 0,C 180,E1 -1761.7,E2 -1761.7} C_VEL
LIN {X 0,Y 580.398,Z 131.522,A -85,B 0,C 180,E1 -1764.464,E2 -1764.464} C_VEL
LIN {X 0,Y 580.312,Z 121.198,A -85,B 0,C 180,E1 -1766.409,E2 -1766.409} C_VEL
LIN {X 0,Y 580.278,Z 121.207,A -85,B 0,C 180,E1 -1769.308,E2 -1769.308} C_VEL
LIN {X 0,Y 580.293,Z 121.197,A -85,B 0,C 180,E1 -1772.143,E2 -1772.143} C_VEL
LIN {X 0,Y 580.289,Z 121.203,A -85,B 0,C 180,E1 -1774.92,E2 -1774.92} C_VEL
LIN {X 0,Y 580.257,Z 121.201,A -85,B 0,C 180,E1 -1777.947,E2 -1777.947} C_VEL
LIN {X 0,Y 580.295,Z 121.205,A -85,B 0,C 180,E1 -1780.914,E2 -1780.914} C_VEL
LIN {X 0,Y 580.261,Z 121.2,A -85,B 0,C 180,E1 -1783.825,E2 -1783.825} C_VEL
LIN {X 0,Y 580.309,Z 121.195,A -85,B 0,C 180,E1 -1785.983,E2 -1785.983} C_VEL
LIN {X 0,Y 580.31,Z 121.201,A -85,B 0,C 180,E1 -1788.827,E2 -1788.827} C_VEL
LIN {X 0,Y 580.305,Z 121.195,A -85,B 0,C 180,E1 -1791.644,E2 -1791.644} C_VEL
LIN {X 0,Y 580.313,Z 121.204,A -85,B 0,C 180,E1 -1794.441,E2 -1794.441} C_VEL
LIN {X 0,Y 580.341,Z 121.194,A -85,B 0,C 180,E1 -1797.918,E2 -1797.918} C_VEL
LIN {X 0,Y 580.265,Z 121.202,A -85,B 0,C 180,E1 -1800.694,E2 -1800.694} C_VEL
LIN {X 0,Y 580.31,Z 121.194,A -85,B 0,C 180,E1 -1802.777,E2 -1802.777} C_VEL
LIN {X 0,Y 580.299,Z 121.198,A -85,B 0,C 180,E1 -1805.56,E2 -1805.56} C_VEL
LIN {X 0,Y 580.295,Z 121.199,A -85,B 0,C 180,E1 -1808.357,E2 -1808.357} C_VEL
LIN {X 0,Y 580.273,Z 121.198,A -85,B 0,C 180,E1 -1811.174,E2 -1811.174} C_VEL
LIN {X 0,Y 580.272,Z 121.199,A -85,B 0,C 180,E1 -1814.319,E2 -1814.319} C_VEL
LIN {X 0,Y 580.228,Z 121.205,A -85,B 0,C 180,E1 -1816.9,E2 -1816.9} C_VEL
LIN {X 0,Y 580.246,Z 121.206,A -85,B 0,C 180,E1 -1819.825,E2 -1819.825} C_VEL
LIN {X 0,Y 580.217,Z 121.207,A -85,B 0,C 180,E1 -1822.055,E2 -1822.055} C_VEL
LIN {X 0,Y 580.247,Z 121.203,A -85,B 0,C 180,E1 -1824.713,E2 -1824.713} C_VEL
LIN {X 0,Y 580.249,Z 121.208,A -85,B 0,C 180,E1 -1827.404,E2 -1827.404} C_VEL
LIN {X 0,Y 580.25,Z 121.203,A -85,B 0,C 180,E1 -1829.775,E2 -1829.775} C_VEL
LIN {X 0,Y 580.287,Z 121.196,A -85,B 0,C 180,E1 -1832.202,E2 -1832.202} C_VEL
LIN {X 0,Y 580.279,Z 121.203,A -85,B 0,C 180,E1 -1834.697,E2 -1834.697} C_VEL
LIN {X 0,Y 580.289,Z 121.2,A -85,B 0,C 180,E1 -1837.27,E2 -1837.27} C_VEL
LIN {X 0,Y 580.285,Z 121.2,A -85,B 0,C 180,E1 -1840.269,E2 -1840.269} C_VEL
LIN {X 0,Y 580.26,Z 121.21,A -85,B 0,C 180,E1 -1842.708,E2 -1842.708} C_VEL
LIN {X 0,Y 580.255,Z 121.201,A -85,B 0,C 180,E1 -1845.611,E2 -1845.611} C_VEL
LIN {X 0,Y 580.277,Z 121.205,A -85,B 0,C 180,E1 -1848.67,E2 -1848.67} C_VEL
LIN {X 0,Y 580.273,Z 121.201,A -85,B 0,C 180,E1 -1850.964,E2 -1850.964} C_VEL
LIN {X 0,Y 580.252,Z 121.202,A -85,B 0,C 180,E1 -1853.595,E2 -1853.595} C_VEL
LIN {X 0,Y 580.315,Z 121.203,A -85,B 0,C 180,E1 -1856.145,E2 -1856.145} C_VEL
LIN {X 0,Y 580.272,Z 121.202,A -85,B 0,C 180,E1 -1858.614,E2 -1858.614} C_VEL
LIN {X 0,Y 580.29,Z 121.197,A -85,B 0,C 180,E1 -1861.023,E2 -1861.023} C_VEL
LIN {X 0,Y 580.271,Z 121.206,A -85,B 0,C 180,E1 -1863.671,E2 -1863.671} C_VEL
LIN {X 0,Y 580.316,Z 121.216,A -85,B 0,C 180,E1 -1866.325,E2 -1866.325} C_VEL
LIN {X 0,Y 580.912,Z 125.704,A -85,B 0,C 180,E1 -1866.964,E2 -1866.964} C_VEL
LIN {X 0,Y 580.816,Z 145.339,A -85,B 0,C 180,E1 -1869.642,E2 -1869.642} C_VEL
LIN {X 0,Y 580.625,Z 165.35,A -85,B 0,C 180,E1 -1872.385,E2 -1872.385} C_VEL
LIN {X 0,Y 580.457,Z 185.294,A -85,B 0,C 180,E1 -1875.09,E2 -1875.09} C_VEL
LIN {X 0,Y 580.408,Z 194.518,A -85,B 0,C 180,E1 -1876.331,E2 -1876.331} C_VEL
LIN {X 0,Y 580.965,Z 200.473,A -85,B 0,C 180,E1 -1876.422,E2 -1876.422} C_VEL
LIN {X 0,Y 580.785,Z 302.924,A -85,B 0,C 180,E1 -1877.707,E2 -1877.707} C_VEL
LIN {X 0,Y 580.727,Z 316.204,A -85,B 0,C 180,E1 -1878.016,E2 -1878.016} C_VEL
LIN {X 0,Y 580.674,Z 328.364,A -85,B 0,C 180,E1 -1878.436,E2 -1878.436} C_VEL
LIN {X 0,Y 580.56,Z 340.62,A -85,B 0,C 180,E1 -1879.008,E2 -1879.008} C_VEL
LIN {X 0,Y 580.441,Z 352.195,A -85,B 0,C 180,E1 -1879.712,E2 -1879.712} C_VEL
LIN {X 0,Y 580.346,Z 362.596,A -85,B 0,C 180,E1 -1880.502,E2 -1880.502} C_VEL
LIN {X 0,Y 580.272,Z 371.108,A -85,B 0,C 180,E1 -1881.292,E2 -1881.292} C_VEL
LIN {X 0,Y 580.222,Z 378.957,A -85,B 0,C 180,E1 -1882.168,E2 -1882.168} C_VEL
LIN {X 0,Y 580.154,Z 386.649,A -85,B 0,C 180,E1 -1883.221,E2 -1883.221} C_VEL
LIN {X 0,Y 580.139,Z 393.678,A -85,B 0,C 180,E1 -1884.438,E2 -1884.438} C_VEL
LIN {X 0,Y 580.108,Z 398.37,A -85,B 0,C 180,E1 -1885.483,E2 -1885.483} C_VEL
LIN {X 0,Y 580.123,Z 401.956,A -85,B 0,C 180,E1 -1886.527,E2 -1886.527} C_VEL
LIN {X 0,Y 580.043,Z 403.807,A -85,B 0,C 180,E1 -1887.222,E2 -1887.222} C_VEL
LIN {X 0,Y 580.04,Z 405.197,A -85,B 0,C 180,E1 -1887.916,E2 -1887.916} C_VEL
LIN {X 0,Y 580.04,Z 406.785,A -85,B 0,C 180,E1 -1889.305,E2 -1889.305} C_VEL
LIN {X 0,Y 580.037,Z 407,A -85,B 0,C 180,E1 -1890,E2 -1890} C_VEL
LIN {X 0,Y 580.047,Z 406.187,A -85,B 0,C 180,E1 -1891.388,E2 -1891.388} C_VEL
LIN {X 0,Y 580.04,Z 405.2,A -85,B 0,C 180,E1 -1892.083,E2 -1892.083} C_VEL
LIN {X 0,Y 580.043,Z 403.811,A -85,B 0,C 180,E1 -1892.778,E2 -1892.778} C_VEL
LIN {X 0,Y 580.11,Z 400.897,A -85,B 0,C 180,E1 -1893.82,E2 -1893.82} C_VEL
LIN {X 0,Y 580.053,Z 396.951,A -85,B 0,C 180,E1 -1894.865,E2 -1894.865} C_VEL
LIN {X 0,Y 580.139,Z 390.879,A -85,B 0,C 180,E1 -1896.084,E2 -1896.084} C_VEL
LIN {X 0,Y 580.184,Z 384.24,A -85,B 0,C 180,E1 -1897.132,E2 -1897.132} C_VEL
LIN {X 0,Y 580.25,Z 375.994,A -85,B 0,C 180,E1 -1898.181,E2 -1898.181} C_VEL
LIN {X 0,Y 580.308,Z 367.543,A -85,B 0,C 180,E1 -1899.058,E2 -1899.058} C_VEL
LIN {X 0,Y 580.422,Z 357.103,A -85,B 0,C 180,E1 -1899.935,E2 -1899.935} C_VEL
LIN {X 0,Y 580.506,Z 346.76,A -85,B 0,C 180,E1 -1900.639,E2 -1900.639} C_VEL
LIN {X 0,Y 580.596,Z 335.254,A -85,B 0,C 180,E1 -1901.263,E2 -1901.263} C_VEL
LIN {X 0,Y 580.682,Z 322.483,A -85,B 0,C 180,E1 -1901.784,E2 -1901.784} C_VEL
LIN {X 0,Y 580.777,Z 309.449,A -85,B 0,C 180,E1 -1902.159,E2 -1902.159} C_VEL
LIN {X 0,Y 580.838,Z 297.113,A -85,B 0,C 180,E1 -1902.379,E2 -1902.379} C_VEL
LIN {X 0,Y 580.802,Z 197.411,A -85,B 0,C 180,E1 -1903.62,E2 -1903.62} C_VEL
LIN {X 0,Y 580.413,Z 194.441,A -85,B 0,C 180,E1 -1903.679,E2 -1903.679} C_VEL
LIN {X 0,Y 580.571,Z 172.004,A -85,B 0,C 180,E1 -1906.708,E2 -1906.708} C_VEL
LIN {X 0,Y 580.727,Z 153.273,A -85,B 0,C 180,E1 -1909.271,E2 -1909.271} C_VEL
LIN {X 0,Y 580.93,Z 133.159,A -85,B 0,C 180,E1 -1912.026,E2 -1912.026} C_VEL
LIN {X 0,Y 580.838,Z 124.063,A -85,B 0,C 180,E1 -1913.287,E2 -1913.287} C_VEL
LIN {X 0,Y 580.296,Z 121.204,A -85,B 0,C 180,E1 -1913.723,E2 -1913.723} C_VEL
LIN {X 0,Y 580.292,Z 121.204,A -85,B 0,C 180,E1 -1916.333,E2 -1916.333} C_VEL
LIN {X 0,Y 580.298,Z 121.196,A -85,B 0,C 180,E1 -1919.308,E2 -1919.308} C_VEL
LIN {X 0,Y 580.297,Z 121.202,A -85,B 0,C 180,E1 -1922.2,E2 -1922.2} C_VEL
LIN {X 0,Y 580.288,Z 121.197,A -85,B 0,C 180,E1 -1924.696,E2 -1924.696} C_VEL
LIN {X 0,Y 580.299,Z 121.196,A -85,B 0,C 180,E1 -1927.268,E2 -1927.268} C_VEL
LIN {X 0,Y 580.296,Z 121.199,A -85,B 0,C 180,E1 -1930.27,E2 -1930.27} C_VEL
LIN {X 0,Y 580.277,Z 121.198,A -85,B 0,C 180,E1 -1932.706,E2 -1932.706} C_VEL
LIN {X 0,Y 580.27,Z 121.206,A -85,B 0,C 180,E1 -1935.609,E2 -1935.609} C_VEL
LIN {X 0,Y 580.299,Z 121.197,A -85,B 0,C 180,E1 -1938.232,E2 -1938.232} C_VEL
LIN {X 0,Y 580.278,Z 121.198,A -85,B 0,C 180,E1 -1940.965,E2 -1940.965} C_VEL
LIN {X 0,Y 580.268,Z 121.209,A -85,B 0,C 180,E1 -1943.596,E2 -1943.596} C_VEL
LIN {X 0,Y 580.3,Z 121.196,A -85,B 0,C 180,E1 -1946.144,E2 -1946.144} C_VEL
LIN {X 0,Y 580.274,Z 121.198,A -85,B 0,C 180,E1 -1948.614,E2 -1948.614} C_VEL
LIN {X 0,Y 580.291,Z 121.199,A -85,B 0,C 180,E1 -1951.023,E2 -1951.023} C_VEL
LIN {X 0,Y 580.29,Z 121.201,A -85,B 0,C 180,E1 -1953.666,E2 -1953.666} C_VEL
LIN {X 0,Y 580.295,Z 121.2,A -85,B 0,C 180,E1 -1955.683,E2 -1955.683} C_VEL
LIN {X 0,Y 580.271,Z 121.199,A -85,B 0,C 180,E1 -1957.947,E2 -1957.947} C_VEL
LIN {X 0,Y 580.298,Z 121.2,A -85,B 0,C 180,E1 -1960.913,E2 -1960.913} C_VEL
LIN {X 0,Y 580.274,Z 121.199,A -85,B 0,C 180,E1 -1963.825,E2 -1963.825} C_VEL
LIN {X 0,Y 580.325,Z 121.192,A -85,B 0,C 180,E1 -1965.983,E2 -1965.983} C_VEL
LIN {X 0,Y 580.304,Z 121.2,A -85,B 0,C 180,E1 -1968.827,E2 -1968.827} C_VEL
LIN {X 0,Y 580.325,Z 121.193,A -85,B 0,C 180,E1 -1971.644,E2 -1971.644} C_VEL
LIN {X 0,Y 580.331,Z 121.193,A -85,B 0,C 180,E1 -1974.44,E2 -1974.44} C_VEL
LIN {X 0,Y 580.333,Z 121.195,A -85,B 0,C 180,E1 -1977.223,E2 -1977.223} C_VEL
LIN {X 0,Y 580.352,Z 121.188,A -85,B 0,C 180,E1 -1980,E2 -1980} C_VEL
LIN {X 0,Y 580.339,Z 121.2,A -85,B 0,C 180,E1 -1982.776,E2 -1982.776} C_VEL
LIN {X 0,Y 580.325,Z 121.192,A -85,B 0,C 180,E1 -1985.559,E2 -1985.559} C_VEL
LIN {X 0,Y 580.333,Z 121.195,A -85,B 0,C 180,E1 -1988.356,E2 -1988.356} C_VEL
LIN {X 0,Y 580.298,Z 121.197,A -85,B 0,C 180,E1 -1991.191,E2 -1991.191} C_VEL
LIN {X 0,Y 580.323,Z 121.194,A -85,B 0,C 180,E1 -1994.017,E2 -1994.017} C_VEL
LIN {X 0,Y 580.309,Z 121.197,A -85,B 0,C 180,E1 -1996.913,E2 -1996.913} C_VEL
LIN {X 0,Y 580.303,Z 121.196,A -85,B 0,C 180,E1 -1999.822,E2 -1999.822} C_VEL
LIN {X 0,Y 580.28,Z 121.197,A -85,B 0,C 180,E1 -2001.333,E2 -2001.333} C_VEL
LIN {X 0,Y 579.584,Z 121.288,A -85,B 0,C 180,E1 -2001.913,E2 -2001.913} C_VEL
LIN {X 0,Y 576.708,Z 121.645,A -85,B 0,C 180,E1 -2002.852,E2 -2002.852} C_VEL
LIN {X 0,Y 574.313,Z 121.942,A -85,B 0,C 180,E1 -2003.609,E2 -2003.609} C_VEL
LIN {X 0,Y 573.314,Z 122.072,A -85,B 0,C 180,E1 -2004.193,E2 -2004.193} C_VEL
LIN {X 0,Y 573.247,Z 122.076,A -85,B 0,C 180,E1 -2004.39,E2 -2004.39} C_VEL
LIN {X 0,Y 573.261,Z 122.072,A -85,B 0,C 180,E1 -2006.975,E2 -2006.975} C_VEL
LIN {X 0,Y 573.244,Z 122.074,A -85,B 0,C 180,E1 -2009.488,E2 -2009.488} C_VEL
LIN {X 0,Y 573.252,Z 122.082,A -85,B 0,C 180,E1 -2012.229,E2 -2012.229} C_VEL
LIN {X 0,Y 573.236,Z 122.076,A -85,B 0,C 180,E1 -2014.772,E2 -2014.772} C_VEL
LIN {X 0,Y 573.251,Z 122.073,A -85,B 0,C 180,E1 -2017.166,E2 -2017.166} C_VEL
LIN {X 0,Y 573.245,Z 122.077,A -85,B 0,C 180,E1 -2019.607,E2 -2019.607} C_VEL
LIN {X 0,Y 573.239,Z 122.075,A -85,B 0,C 180,E1 -2022.642,E2 -2022.642} C_VEL
LIN {X 0,Y 573.235,Z 122.081,A -85,B 0,C 180,E1 -2025.667,E2 -2025.667} C_VEL
LIN {X 0,Y 573.241,Z 122.075,A -85,B 0,C 180,E1 -2028.544,E2 -2028.544} C_VEL
LIN {X 0,Y 573.246,Z 122.076,A -85,B 0,C 180,E1 -2031.299,E2 -2031.299} C_VEL
LIN {X 0,Y 573.24,Z 122.079,A -85,B 0,C 180,E1 -2034.014,E2 -2034.014} C_VEL
LIN {X 0,Y 573.281,Z 122.069,A -85,B 0,C 180,E1 -2036.519,E2 -2036.519} C_VEL
LIN {X 0,Y 573.234,Z 122.077,A -85,B 0,C 180,E1 -2039.116,E2 -2039.116} C_VEL
LIN {X 0,Y 573.261,Z 122.075,A -85,B 0,C 180,E1 -2041.968,E2 -2041.968} C_VEL
LIN {X 0,Y 573.251,Z 122.073,A -85,B 0,C 180,E1 -2044.59,E2 -2044.59} C_VEL
LIN {X 0,Y 573.234,Z 122.081,A -85,B 0,C 180,E1 -2047.663,E2 -2047.663} C_VEL
LIN {X 0,Y 573.273,Z 122.071,A -85,B 0,C 180,E1 -2050.671,E2 -2050.671} C_VEL
LIN {X 0,Y 573.248,Z 122.078,A -85,B 0,C 180,E1 -2053.622,E2 -2053.622} C_VEL
LIN {X 0,Y 573.269,Z 122.073,A -85,B 0,C 180,E1 -2055.807,E2 -2055.807} C_VEL
LIN {X 0,Y 573.259,Z 122.074,A -85,B 0,C 180,E1 -2058.745,E2 -2058.745} C_VEL
LIN {X 0,Y 573.287,Z 122.072,A -85,B 0,C 180,E1 -2061.541,E2 -2061.541} C_VEL
LIN {X 0,Y 573.297,Z 122.068,A -85,B 0,C 180,E1 -2064.372,E2 -2064.372} C_VEL
LIN {X 0,Y 573.314,Z 122.065,A -85,B 0,C 180,E1 -2067.893,E2 -2067.893} C_VEL
LIN {X 0,Y 573.329,Z 122.068,A -85,B 0,C 180,E1 -2070.703,E2 -2070.703} C_VEL
LIN {X 0,Y 573.303,Z 122.074,A -85,B 0,C 180,E1 -2072.811,E2 -2072.811} C_VEL
LIN {X 0,Y 573.297,Z 122.068,A -85,B 0,C 180,E1 -2075.629,E2 -2075.629} C_VEL
LIN {X 0,Y 573.287,Z 122.072,A -85,B 0,C 180,E1 -2078.46,E2 -2078.46} C_VEL
LIN {X 0,Y 573.269,Z 122.073,A -85,B 0,C 180,E1 -2081.312,E2 -2081.312} C_VEL
LIN {X 0,Y 573.279,Z 122.075,A -85,B 0,C 180,E1 -2084.425,E2 -2084.425} C_VEL
LIN {X 0,Y 573.257,Z 122.076,A -85,B 0,C 180,E1 -2087.112,E2 -2087.112} C_VEL
LIN {X 0,Y 573.29,Z 122.145,A -85,B 0,C 180,E1 -2089.656,E2 -2089.656} C_VEL
LIN {X 0,Y 573.366,Z 134.38,A -85,B 0,C 180,E1 -2091.954,E2 -2091.954} C_VEL
LIN {X 0,Y 573.237,Z 146.628,A -85,B 0,C 180,E1 -2094.226,E2 -2094.226} C_VEL
LIN {X 0,Y 574.071,Z 153.025,A -85,B 0,C 180,E1 -2094.333,E2 -2094.333} C_VEL
LIN {X 0,Y 573.82,Z 253.008,A -85,B 0,C 180,E1 -2095.602,E2 -2095.602} C_VEL
LIN {X 0,Y 573.751,Z 266.495,A -85,B 0,C 180,E1 -2095.922,E2 -2095.922} C_VEL
LIN {X 0,Y 573.64,Z 278.82,A -85,B 0,C 180,E1 -2096.356,E2 -2096.356} C_VEL
LIN {X 0,Y 573.563,Z 290.34,A -85,B 0,C 180,E1 -2096.902,E2 -2096.902} C_VEL
LIN {X 0,Y 573.44,Z 301.172,A -85,B 0,C 180,E1 -2097.559,E2 -2097.559} C_VEL
LIN {X 0,Y 573.322,Z 312.414,A -85,B 0,C 180,E1 -2098.415,E2 -2098.415} C_VEL
LIN {X 0,Y 573.239,Z 320.483,A -85,B 0,C 180,E1 -2099.166,E2 -2099.166} C_VEL
LIN {X 0,Y 573.161,Z 329.478,A -85,B 0,C 180,E1 -2100.182,E2 -2100.182} C_VEL
LIN {X 0,Y 573.077,Z 336.813,A -85,B 0,C 180,E1 -2101.208,E2 -2101.208} C_VEL
LIN {X 0,Y 573.039,Z 343.617,A -85,B 0,C 180,E1 -2102.402,E2 -2102.402} C_VEL
LIN {X 0,Y 572.991,Z 348.488,A -85,B 0,C 180,E1 -2103.501,E2 -2103.501} C_VEL
LIN {X 0,Y 572.987,Z 352.559,A -85,B 0,C 180,E1 -2104.736,E2 -2104.736} C_VEL
LIN {X 0,Y 572.921,Z 355.418,A -85,B 0,C 180,E1 -2106.073,E2 -2106.073} C_VEL
LIN {X 0,Y 572.926,Z 356.638,A -85,B 0,C 180,E1 -2107.123,E2 -2107.123} C_VEL
LIN {X 0,Y 572.928,Z 356.956,A -85,B 0,C 180,E1 -2108.273,E2 -2108.273} C_VEL
LIN {X 0,Y 572.925,Z 355.975,A -85,B 0,C 180,E1 -2109.634,E2 -2109.634} C_VEL
LIN {X 0,Y 572.938,Z 353.413,A -85,B 0,C 180,E1 -2111.016,E2 -2111.016} C_VEL
LIN {X 0,Y 573.01,Z 350.724,A -85,B 0,C 180,E1 -2111.966,E2 -2111.966} C_VEL
LIN {X 0,Y 573.021,Z 346.944,A -85,B 0,C 180,E1 -2112.972,E2 -2112.972} C_VEL
LIN {X 0,Y 573.061,Z 341.131,A -85,B 0,C 180,E1 -2114.16,E2 -2114.16} C_VEL
LIN {X 0,Y 573.096,Z 333.732,A -85,B 0,C 180,E1 -2115.339,E2 -2115.339} C_VEL
LIN {X 0,Y 573.177,Z 325.905,A -85,B 0,C 180,E1 -2116.339,E2 -2116.339} C_VEL
LIN {X 0,Y 573.285,Z 317.466,A -85,B 0,C 180,E1 -2117.222,E2 -2117.222} C_VEL
LIN {X 0,Y 573.369,Z 306.692,A -85,B 0,C 180,E1 -2118.135,E2 -2118.135} C_VEL
LIN {X 0,Y 573.473,Z 295.212,A -85,B 0,C 180,E1 -2118.913,E2 -2118.913} C_VEL
LIN {X 0,Y 573.621,Z 283.963,A -85,B 0,C 180,E1 -2119.508,E2 -2119.508} C_VEL
LIN {X 0,Y 573.758,Z 270.674,A -85,B 0,C 180,E1 -2120.036,E2 -2120.036} C_VEL
LIN {X 0,Y 573.808,Z 258.264,A -85,B 0,C 180,E1 -2120.383,E2 -2120.383} C_VEL
LIN {X 0,Y 573.853,Z 245.398,A -85,B 0,C 180,E1 -2120.599,E2 -2120.599} C_VEL
LIN {X 0,Y 573.96,Z 151.118,A -85,B 0,C 180,E1 -2121.784,E2 -2121.784} C_VEL
LIN {X 0,Y 573.217,Z 146.632,A -85,B 0,C 180,E1 -2121.863,E2 -2121.863} C_VEL
LIN {X 0,Y 573.368,Z 131.796,A -85,B 0,C 180,E1 -2124.619,E2 -2124.619} C_VEL
LIN {X 0,Y 573.279,Z 122.075,A -85,B 0,C 180,E1 -2126.424,E2 -2126.424} C_VEL
LIN {X 0,Y 573.226,Z 122.084,A -85,B 0,C 180,E1 -2129.119,E2 -2129.119} C_VEL
LIN {X 0,Y 573.237,Z 122.083,A -85,B 0,C 180,E1 -2131.436,E2 -2131.436} C_VEL
LIN {X 0,Y 573.261,Z 122.075,A -85,B 0,C 180,E1 -2133.811,E2 -2133.811} C_VEL
LIN {X 0,Y 573.213,Z 122.079,A -85,B 0,C 180,E1 -2136.134,E2 -2136.134} C_VEL
LIN {X 0,Y 573.25,Z 122.081,A -85,B 0,C 180,E1 -2139.174,E2 -2139.174} C_VEL
LIN {X 0,Y 573.212,Z 122.081,A -85,B 0,C 180,E1 -2141.411,E2 -2141.411} C_VEL
LIN {X 0,Y 573.239,Z 122.076,A -85,B 0,C 180,E1 -2143.622,E2 -2143.622} C_VEL
LIN {X 0,Y 573.254,Z 122.073,A -85,B 0,C 180,E1 -2145.807,E2 -2145.807} C_VEL
LIN {X 0,Y 573.268,Z 122.08,A -85,B 0,C 180,E1 -2148.746,E2 -2148.746} C_VEL
LIN {X 0,Y 573.249,Z 122.074,A -85,B 0,C 180,E1 -2151.54,E2 -2151.54} C_VEL
LIN {X 0,Y 573.281,Z 122.078,A -85,B 0,C 180,E1 -2154.372,E2 -2154.372} C_VEL
LIN {X 0,Y 573.311,Z 122.069,A -85,B 0,C 180,E1 -2157.893,E2 -2157.893} C_VEL
LIN {X 0,Y 573.32,Z 122.069,A -85,B 0,C 180,E1 -2160,E2 -2160} C_VEL
LIN {X 0,Y 573.277,Z 122.07,A -85,B 0,C 180,E1 -2162.811,E2 -2162.811} C_VEL
LIN {X 0,Y 573.268,Z 122.075,A -85,B 0,C 180,E1 -2165.629,E2 -2165.629} C_VEL
LIN {X 0,Y 573.236,Z 122.077,A -85,B 0,C 180,E1 -2168.461,E2 -2168.461} C_VEL
LIN {X 0,Y 573.241,Z 122.075,A -85,B 0,C 180,E1 -2171.313,E2 -2171.313} C_VEL
LIN {X 0,Y 573.23,Z 122.076,A -85,B 0,C 180,E1 -2174.402,E2 -2174.402} C_VEL
LIN {X 0,Y 573.178,Z 122.084,A -85,B 0,C 180,E1 -2177.114,E2 -2177.114} C_VEL
LIN {X 0,Y 573.19,Z 122.082,A -85,B 0,C 180,E1 -2180.079,E2 -2180.079} C_VEL
LIN {X 0,Y 573.19,Z 122.081,A -85,B 0,C 180,E1 -2182.34,E2 -2182.34} C_VEL
LIN {X 0,Y 573.197,Z 122.082,A -85,B 0,C 180,E1 -2184.862,E2 -2184.862} C_VEL
LIN {X 0,Y 573.19,Z 122.086,A -85,B 0,C 180,E1 -2186.979,E2 -2186.979} C_VEL
LIN {X 0,Y 573.201,Z 122.084,A -85,B 0,C 180,E1 -2189.479,E2 -2189.479} C_VEL
LIN {X 0,Y 573.241,Z 122.074,A -85,B 0,C 180,E1 -2192.225,E2 -2192.225} C_VEL
LIN {X 0,Y 573.225,Z 122.083,A -85,B 0,C 180,E1 -2194.769,E2 -2194.769} C_VEL
LIN {X 0,Y 573.23,Z 122.076,A -85,B 0,C 180,E1 -2197.808,E2 -2197.808} C_VEL
LIN {X 0,Y 573.251,Z 122.079,A -85,B 0,C 180,E1 -2200.525,E2 -2200.525} C_VEL
LIN {X 0,Y 573.211,Z 122.078,A -85,B 0,C 180,E1 -2203.665,E2 -2203.665} C_VEL
LIN {X 0,Y 573.207,Z 122.088,A -85,B 0,C 180,E1 -2206.637,E2 -2206.637} C_VEL
LIN {X 0,Y 573.25,Z 122.074,A -85,B 0,C 180,E1 -2209.475,E2 -2209.475} C_VEL
LIN {X 0,Y 573.233,Z 122.083,A -85,B 0,C 180,E1 -2212.192,E2 -2212.192} C_VEL
LIN {X 0,Y 573.236,Z 122.075,A -85,B 0,C 180,E1 -2215.229,E2 -2215.229} C_VEL
LIN {X 0,Y 573.251,Z 122.079,A -85,B 0,C 180,E1 -2217.772,E2 -2217.772} C_VEL
LIN {X 0,Y 573.247,Z 122.076,A -85,B 0,C 180,E1 -2220.633,E2 -2220.633} C_VEL
LIN {X 0,Y 573.213,Z 122.079,A -85,B 0,C 180,E1 -2223.022,E2 -2223.022} C_VEL
LIN {X 0,Y 573.28,Z 122.074,A -85,B 0,C 180,E1 -2225.366,E2 -2225.366} C_VEL
LIN {X 0,Y 573.265,Z 122.145,A -85,B 0,C 180,E1 -2226.202,E2 -2226.202} C_VEL
LIN {X 0,Y 573.953,Z 127.186,A -85,B 0,C 180,E1 -2226.931,E2 -2226.931} C_VEL
LIN {X 0,Y 573.821,Z 146.31,A -85,B 0,C 180,E1 -2229.57,E2 -2229.57} C_VEL
LIN {X 0,Y 573.658,Z 166.813,A -85,B 0,C 180,E1 -2232.367,E2 -2232.367} C_VEL
LIN {X 0,Y 573.452,Z 186.624,A -85,B 0,C 180,E1 -2235.086,E2 -2235.086} C_VEL
LIN {X 0,Y 573.398,Z 194.518,A -85,B 0,C 180,E1 -2236.16,E2 -2236.16} C_VEL
LIN {X 0,Y 574.059,Z 200.473,A -85,B 0,C 180,E1 -2236.256,E2 -2236.256} C_VEL
LIN {X 0,Y 573.85,Z 302.924,A -85,B 0,C 180,E1 -2237.556,E2 -2237.556} C_VEL
LIN {X 0,Y 573.779,Z 316.203,A -85,B 0,C 180,E1 -2237.869,E2 -2237.869} C_VEL
LIN {X 0,Y 573.7,Z 328.366,A -85,B 0,C 180,E1 -2238.294,E2 -2238.294} C_VEL
LIN {X 0,Y 573.567,Z 340.621,A -85,B 0,C 180,E1 -2238.873,E2 -2238.873} C_VEL
LIN {X 0,Y 573.428,Z 352.192,A -85,B 0,C 180,E1 -2239.585,E2 -2239.585} C_VEL
LIN {X 0,Y 573.333,Z 362.598,A -85,B 0,C 180,E1 -2240.385,E2 -2240.385} C_VEL
LIN {X 0,Y 573.241,Z 371.109,A -85,B 0,C 180,E1 -2241.184,E2 -2241.184} C_VEL
LIN {X 0,Y 573.161,Z 378.957,A -85,B 0,C 180,E1 -2242.071,E2 -2242.071} C_VEL
LIN {X 0,Y 573.073,Z 386.953,A -85,B 0,C 180,E1 -2243.185,E2 -2243.185} C_VEL
LIN {X 0,Y 573.071,Z 393.678,A -85,B 0,C 180,E1 -2244.369,E2 -2244.369} C_VEL
LIN {X 0,Y 573.029,Z 398.371,A -85,B 0,C 180,E1 -2245.427,E2 -2245.427} C_VEL
LIN {X 0,Y 573.022,Z 401.956,A -85,B 0,C 180,E1 -2246.484,E2 -2246.484} C_VEL
LIN {X 0,Y 572.959,Z 403.807,A -85,B 0,C 180,E1 -2247.187,E2 -2247.187} C_VEL
LIN {X 0,Y 572.946,Z 406.184,A -85,B 0,C 180,E1 -2248.594,E2 -2248.594} C_VEL
LIN {X 0,Y 572.938,Z 407,A -85,B 0,C 180,E1 -2250,E2 -2250} C_VEL
LIN {X 0,Y 572.946,Z 406.186,A -85,B 0,C 180,E1 -2251.405,E2 -2251.405} C_VEL
LIN {X 0,Y 572.94,Z 405.199,A -85,B 0,C 180,E1 -2252.109,E2 -2252.109} C_VEL
LIN {X 0,Y 572.959,Z 403.811,A -85,B 0,C 180,E1 -2252.812,E2 -2252.812} C_VEL
LIN {X 0,Y 573.014,Z 400.897,A -85,B 0,C 180,E1 -2253.868,E2 -2253.868} C_VEL
LIN {X 0,Y 572.963,Z 396.95,A -85,B 0,C 180,E1 -2254.925,E2 -2254.925} C_VEL
LIN {X 0,Y 573.093,Z 391.869,A -85,B 0,C 180,E1 -2255.983,E2 -2255.983} C_VEL
LIN {X 0,Y 573.103,Z 385.471,A -85,B 0,C 180,E1 -2257.044,E2 -2257.044} C_VEL
LIN {X 0,Y 573.177,Z 377.481,A -85,B 0,C 180,E1 -2258.106,E2 -2258.106} C_VEL
LIN {X 0,Y 573.254,Z 369.339,A -85,B 0,C 180,E1 -2258.993,E2 -2258.993} C_VEL
LIN {X 0,Y 573.348,Z 359.404,A -85,B 0,C 180,E1 -2259.881,E2 -2259.881} C_VEL
LIN {X 0,Y 573.512,Z 348.219,A -85,B 0,C 180,E1 -2260.679,E2 -2260.679} C_VEL
LIN {X 0,Y 573.586,Z 337.182,A -85,B 0,C 180,E1 -2261.305,E2 -2261.305} C_VEL
LIN {X 0,Y 573.708,Z 324.991,A -85,B 0,C 180,E1 -2261.84,E2 -2261.84} C_VEL
LIN {X 0,Y 573.838,Z 312.191,A -85,B 0,C 180,E1 -2262.241,E2 -2262.241} C_VEL
LIN {X 0,Y 573.88,Z 298.627,A -85,B 0,C 180,E1 -2262.51,E2 -2262.51} C_VEL
LIN {X 0,Y 573.906,Z 198.081,A -85,B 0,C 180,E1 -2263.778,E2 -2263.778} C_VEL
LIN {X 0,Y 573.417,Z 194.441,A -85,B 0,C 180,E1 -2263.85,E2 -2263.85} C_VEL
LIN {X 0,Y 573.582,Z 173.359,A -85,B 0,C 180,E1 -2266.731,E2 -2266.731} C_VEL
LIN {X 0,Y 573.74,Z 153.899,A -85,B 0,C 180,E1 -2269.402,E2 -2269.402} C_VEL
LIN {X 0,Y 573.997,Z 134.226,A -85,B 0,C 180,E1 -2272.117,E2 -2272.117} C_VEL
LIN {X 0,Y 573.922,Z 125.784,A -85,B 0,C 180,E1 -2273.304,E2 -2273.304} C_VEL
LIN {X 0,Y 573.25,Z 122.082,A -85,B 0,C 180,E1 -2273.864,E2 -2273.864} C_VEL
LIN {X 0,Y 573.237,Z 122.08,A -85,B 0,C 180,E1 -2276.492,E2 -2276.492} C_VEL
LIN {X 0,Y 573.262,Z 122.073,A -85,B 0,C 180,E1 -2279.366,E2 -2279.366} C_VEL
LIN {X 0,Y 573.25,Z 122.079,A -85,B 0,C 180,E1 -2282.227,E2 -2282.227} C_VEL
LIN {X 0,Y 573.235,Z 122.075,A -85,B 0,C 180,E1 -2284.771,E2 -2284.771} C_VEL
LIN {X 0,Y 573.236,Z 122.083,A -85,B 0,C 180,E1 -2287.807,E2 -2287.807} C_VEL
LIN {X 0,Y 573.245,Z 122.075,A -85,B 0,C 180,E1 -2290.525,E2 -2290.525} C_VEL
LIN {X 0,Y 573.237,Z 122.078,A -85,B 0,C 180,E1 -2293.359,E2 -2293.359} C_VEL
LIN {X 0,Y 573.245,Z 122.075,A -85,B 0,C 180,E1 -2296.331,E2 -2296.331} C_VEL
LIN {X 0,Y 573.239,Z 122.074,A -85,B 0,C 180,E1 -2298.543,E2 -2298.543} C_VEL
